MoveJ RelTool (starting_position, 122, -10.9, -364 \Rx:=2.5, \Ry:=-2.1, \Rz:=0), v200, z200, Tooldata_7;
MoveJ RelTool (starting_position, 122, -11.6, -364 \Rx:=2.5, \Ry:=-2.1, \Rz:=0), v200, z200, Tooldata_7;
MoveJ RelTool (starting_position, 121, -12.4, -364 \Rx:=2.6, \Ry:=-2.1, \Rz:=0), v200, z200, Tooldata_7;
MoveJ RelTool (starting_position, 120, -13.1, -364 \Rx:=2.6, \Ry:=-2.4, \Rz:=0), v200, z200, Tooldata_7;
MoveJ RelTool (starting_position, 119, -13.8, -364 \Rx:=2.7, \Ry:=-2.4, \Rz:=0), v200, z200, Tooldata_7;
MoveJ RelTool (starting_position, 119, -14.6, -363 \Rx:=2.8, \Ry:=-2.7, \Rz:=0), v200, z200, Tooldata_7;
MoveJ RelTool (starting_position, 118, -15.4, -363 \Rx:=3, \Ry:=-2.7, \Rz:=0), v200, z200, Tooldata_7;
MoveJ RelTool (starting_position, 117, -16.1, -363 \Rx:=3.2, \Ry:=-3, \Rz:=0), v200, z200, Tooldata_7;
MoveJ RelTool (starting_position, 116, -16.9, -363 \Rx:=3.4, \Ry:=-3, \Rz:=0), v200, z200, Tooldata_7;
MoveJ RelTool (starting_position, 115, -17.6, -363 \Rx:=3.6, \Ry:=-3.3, \Rz:=0), v200, z200, Tooldata_7;
MoveJ RelTool (starting_position, 114, -18.3, -363 \Rx:=3.8, \Ry:=-3.3, \Rz:=0), v200, z200, Tooldata_7;
MoveJ RelTool (starting_position, 113, -19.1, -363 \Rx:=4.1, \Ry:=-3.6, \Rz:=0), v200, z200, Tooldata_7;
MoveJ RelTool (starting_position, 112, -19.8, -363 \Rx:=4.3, \Ry:=-3.9, \Rz:=0), v200, z200, Tooldata_7;
MoveJ RelTool (starting_position, 111, -20.5, -362 \Rx:=4.6, \Ry:=-3.9, \Rz:=0), v200, z200, Tooldata_7;
MoveJ RelTool (starting_position, 110, -21.1, -362 \Rx:=4.8, \Ry:=-4.2, \Rz:=0), v200, z200, Tooldata_7;
MoveJ RelTool (starting_position, 109, -21.8, -362 \Rx:=5, \Ry:=-4.2, \Rz:=0), v200, z200, Tooldata_7;
MoveJ RelTool (starting_position, 108, -22.4, -362 \Rx:=5.2, \Ry:=-4.5, \Rz:=0), v200, z200, Tooldata_7;
MoveJ RelTool (starting_position, 107, -23, -361 \Rx:=5.5, \Ry:=-4.5, \Rz:=0), v200, z200, Tooldata_7;
MoveJ RelTool (starting_position, 107, -23.6, -361 \Rx:=5.6, \Ry:=-4.8, \Rz:=0), v200, z200, Tooldata_7;
MoveJ RelTool (starting_position, 106, -24.1, -360 \Rx:=5.8, \Ry:=-4.8, \Rz:=0), v200, z200, Tooldata_7;
MoveJ RelTool (starting_position, 105, -24.6, -360 \Rx:=5.9, \Ry:=-5.1, \Rz:=0), v200, z200, Tooldata_7;
MoveJ RelTool (starting_position, 104, -25.1, -359 \Rx:=6, \Ry:=-5.1, \Rz:=0), v200, z200, Tooldata_7;
MoveJ RelTool (starting_position, 103, -25.6, -359 \Rx:=6.2, \Ry:=-5.4, \Rz:=0), v200, z200, Tooldata_7;
MoveJ RelTool (starting_position, 103, -26, -358 \Rx:=6.3, \Ry:=-5.4, \Rz:=0), v200, z200, Tooldata_7;
MoveJ RelTool (starting_position, 103, -26.4, -357 \Rx:=6.4, \Ry:=-5.4, \Rz:=0), v200, z200, Tooldata_7;
MoveJ RelTool (starting_position, 103, -26.8, -356 \Rx:=6.5, \Ry:=-5.4, \Rz:=0), v200, z200, Tooldata_7;
MoveJ RelTool (starting_position, 103, -27.1, -355 \Rx:=6.6, \Ry:=-5.4, \Rz:=0), v200, z200, Tooldata_7;
MoveJ RelTool (starting_position, 103, -27.5, -354 \Rx:=6.7, \Ry:=-5.4, \Rz:=0), v200, z200, Tooldata_7;
MoveJ RelTool (starting_position, 103, -27.8, -353 \Rx:=6.8, \Ry:=-5.4, \Rz:=0), v200, z200, Tooldata_7;
MoveJ RelTool (starting_position, 103, -28.2, -352 \Rx:=6.9, \Ry:=-5.4, \Rz:=0), v200, z200, Tooldata_7;
MoveJ RelTool (starting_position, 104, -28.5, -351 \Rx:=7, \Ry:=-5.1, \Rz:=0), v200, z200, Tooldata_7;
MoveJ RelTool (starting_position, 105, -28.8, -350 \Rx:=7.1, \Ry:=-5.1, \Rz:=0), v200, z200, Tooldata_7;
MoveJ RelTool (starting_position, 106, -29, -349 \Rx:=7.2, \Ry:=-4.8, \Rz:=0), v200, z200, Tooldata_7;
MoveJ RelTool (starting_position, 108, -29.3, -348 \Rx:=7.4, \Ry:=-4.5, \Rz:=0), v200, z200, Tooldata_7;
MoveJ RelTool (starting_position, 109, -29.6, -347 \Rx:=7.6, \Ry:=-4.2, \Rz:=0), v200, z200, Tooldata_7;
MoveJ RelTool (starting_position, 111, -29.8, -346 \Rx:=7.8, \Ry:=-3.9, \Rz:=0), v200, z200, Tooldata_7;
MoveJ RelTool (starting_position, 113, -30.1, -345 \Rx:=8.1, \Ry:=-3.6, \Rz:=0), v200, z200, Tooldata_7;
MoveJ RelTool (starting_position, 115, -30.4, -344 \Rx:=8.4, \Ry:=-3.3, \Rz:=0), v200, z200, Tooldata_7;
MoveJ RelTool (starting_position, 117, -30.6, -343 \Rx:=8.7, \Ry:=-3, \Rz:=0), v200, z200, Tooldata_7;
MoveJ RelTool (starting_position, 119, -30.9, -343 \Rx:=8.9, \Ry:=-2.7, \Rz:=0), v200, z200, Tooldata_7;
MoveJ RelTool (starting_position, 121, -31.2, -342 \Rx:=9.2, \Ry:=-2.1, \Rz:=0), v200, z200, Tooldata_7;
MoveJ RelTool (starting_position, 123, -31.5, -342 \Rx:=9.5, \Ry:=-1.8, \Rz:=0), v200, z200, Tooldata_7;
MoveJ RelTool (starting_position, 126, -31.8, -341 \Rx:=9.7, \Ry:=-1.5, \Rz:=0), v200, z200, Tooldata_7;
MoveJ RelTool (starting_position, 128, -32.1, -341 \Rx:=10, \Ry:=-0.9, \Rz:=0), v200, z200, Tooldata_7;
MoveJ RelTool (starting_position, 131, -32.4, -341 \Rx:=10.3, \Ry:=-0.6, \Rz:=0), v200, z200, Tooldata_7;
MoveJ RelTool (starting_position, 134, -32.8, -341 \Rx:=10.6, \Ry:=-0, \Rz:=0), v200, z200, Tooldata_7;
MoveJ RelTool (starting_position, 137, -33.2, -341 \Rx:=10.9, \Ry:=0.6, \Rz:=0), v200, z200, Tooldata_7;
MoveJ RelTool (starting_position, 139, -33.6, -341 \Rx:=11.1, \Ry:=0.9, \Rz:=0), v200, z200, Tooldata_7;
MoveJ RelTool (starting_position, 142, -34, -341 \Rx:=11.3, \Ry:=1.5, \Rz:=0), v200, z200, Tooldata_7;
MoveJ RelTool (starting_position, 145, -34.4, -341 \Rx:=11.5, \Ry:=2.1, \Rz:=0), v200, z200, Tooldata_7;
MoveJ RelTool (starting_position, 148, -34.8, -342 \Rx:=11.6, \Ry:=2.4, \Rz:=0), v200, z200, Tooldata_7;
MoveJ RelTool (starting_position, 150, -35.3, -342 \Rx:=11.8, \Ry:=3, \Rz:=0), v200, z200, Tooldata_7;
MoveJ RelTool (starting_position, 153, -35.9, -343 \Rx:=11.9, \Ry:=3.3, \Rz:=0), v200, z200, Tooldata_7;
MoveJ RelTool (starting_position, 155, -36.4, -344 \Rx:=12, \Ry:=3.6, \Rz:=0), v200, z200, Tooldata_7;
MoveJ RelTool (starting_position, 157, -37, -344 \Rx:=12, \Ry:=4.2, \Rz:=0), v200, z200, Tooldata_7;
MoveJ RelTool (starting_position, 159, -37.6, -345 \Rx:=12, \Ry:=4.5, \Rz:=0), v200, z200, Tooldata_7;
MoveJ RelTool (starting_position, 161, -38.2, -346 \Rx:=12, \Ry:=4.8, \Rz:=0), v200, z200, Tooldata_7;
MoveJ RelTool (starting_position, 163, -38.8, -347 \Rx:=12, \Ry:=5.1, \Rz:=0), v200, z200, Tooldata_7;
MoveJ RelTool (starting_position, 165, -39.5, -348 \Rx:=11.9, \Ry:=5.4, \Rz:=0), v200, z200, Tooldata_7;
MoveJ RelTool (starting_position, 167, -40.2, -349 \Rx:=11.8, \Ry:=5.7, \Rz:=0), v200, z200, Tooldata_7;
MoveJ RelTool (starting_position, 168, -40.9, -349 \Rx:=11.6, \Ry:=6, \Rz:=0), v200, z200, Tooldata_7;
MoveJ RelTool (starting_position, 170, -41.6, -350 \Rx:=11.4, \Ry:=6.3, \Rz:=0), v200, z200, Tooldata_7;
MoveJ RelTool (starting_position, 171, -42.4, -351 \Rx:=11.1, \Ry:=6.6, \Rz:=0), v200, z200, Tooldata_7;
MoveJ RelTool (starting_position, 172, -43.1, -352 \Rx:=10.8, \Ry:=6.6, \Rz:=0), v200, z200, Tooldata_7;
MoveJ RelTool (starting_position, 173, -43.8, -353 \Rx:=10.4, \Ry:=6.9, \Rz:=0), v200, z200, Tooldata_7;
MoveJ RelTool (starting_position, 173, -44.6, -354 \Rx:=10.1, \Ry:=6.9, \Rz:=0), v200, z200, Tooldata_7;
MoveJ RelTool (starting_position, 174, -45.4, -355 \Rx:=9.6, \Ry:=6.9, \Rz:=0), v200, z200, Tooldata_7;
MoveJ RelTool (starting_position, 174, -46.1, -356 \Rx:=9.1, \Ry:=6.9, \Rz:=0), v200, z200, Tooldata_7;
MoveJ RelTool (starting_position, 175, -46.9, -357 \Rx:=8.6, \Ry:=7.2, \Rz:=0), v200, z200, Tooldata_7;
MoveJ RelTool (starting_position, 175, -47.6, -357 \Rx:=8.1, \Ry:=7.2, \Rz:=0), v200, z200, Tooldata_7;
MoveJ RelTool (starting_position, 175, -48.3, -358 \Rx:=7.6, \Ry:=7.2, \Rz:=0), v200, z200, Tooldata_7;
MoveJ RelTool (starting_position, 175, -49.1, -359 \Rx:=7, \Ry:=7.2, \Rz:=0), v200, z200, Tooldata_7;
MoveJ RelTool (starting_position, 174, -49.8, -360 \Rx:=6.4, \Ry:=6.9, \Rz:=0), v200, z200, Tooldata_7;
MoveJ RelTool (starting_position, 174, -50.5, -361 \Rx:=5.8, \Ry:=6.9, \Rz:=0), v200, z200, Tooldata_7;
MoveJ RelTool (starting_position, 173, -51.1, -361 \Rx:=5.3, \Ry:=6.9, \Rz:=0), v200, z200, Tooldata_7;
MoveJ RelTool (starting_position, 172, -51.8, -362 \Rx:=4.7, \Ry:=6.6, \Rz:=0), v200, z200, Tooldata_7;
MoveJ RelTool (starting_position, 172, -52.4, -363 \Rx:=4.1, \Ry:=6.6, \Rz:=0), v200, z200, Tooldata_7;
MoveJ RelTool (starting_position, 171, -53, -364 \Rx:=3.6, \Ry:=6.6, \Rz:=0), v200, z200, Tooldata_7;
MoveJ RelTool (starting_position, 170, -53.6, -364 \Rx:=3.1, \Ry:=6.3, \Rz:=0), v200, z200, Tooldata_7;
MoveJ RelTool (starting_position, 169, -54.1, -365 \Rx:=2.6, \Ry:=6.3, \Rz:=0), v200, z200, Tooldata_7;
MoveJ RelTool (starting_position, 168, -54.6, -366 \Rx:=2.2, \Ry:=6, \Rz:=0), v200, z200, Tooldata_7;
MoveJ RelTool (starting_position, 167, -55.1, -367 \Rx:=1.8, \Ry:=5.7, \Rz:=0), v200, z200, Tooldata_7;
MoveJ RelTool (starting_position, 165, -55.6, -367 \Rx:=1.4, \Ry:=5.4, \Rz:=0), v200, z200, Tooldata_7;
MoveJ RelTool (starting_position, 163, -56, -368 \Rx:=1, \Ry:=5.1, \Rz:=0), v200, z200, Tooldata_7;
MoveJ RelTool (starting_position, 162, -56.4, -369 \Rx:=0.7, \Ry:=4.8, \Rz:=0), v200, z200, Tooldata_7;
MoveJ RelTool (starting_position, 160, -56.8, -369 \Rx:=0.4, \Ry:=4.5, \Rz:=0), v200, z200, Tooldata_7;
MoveJ RelTool (starting_position, 158, -57.1, -370 \Rx:=0.2, \Ry:=4.2, \Rz:=0), v200, z200, Tooldata_7;
MoveJ RelTool (starting_position, 156, -57.5, -371 \Rx:=-0, \Ry:=3.9, \Rz:=0), v200, z200, Tooldata_7;
MoveJ RelTool (starting_position, 154, -57.8, -371 \Rx:=-0.2, \Ry:=3.6, \Rz:=0), v200, z200, Tooldata_7;
MoveJ RelTool (starting_position, 152, -58.1, -372 \Rx:=-0.3, \Ry:=3.3, \Rz:=0), v200, z200, Tooldata_7;
MoveJ RelTool (starting_position, 150, -58.4, -372 \Rx:=-0.4, \Ry:=2.7, \Rz:=0), v200, z200, Tooldata_7;
MoveJ RelTool (starting_position, 148, -58.7, -373 \Rx:=-0.4, \Ry:=2.4, \Rz:=0), v200, z200, Tooldata_7;
MoveJ RelTool (starting_position, 145, -59, -373 \Rx:=-0.4, \Ry:=2.1, \Rz:=0), v200, z200, Tooldata_7;
MoveJ RelTool (starting_position, 143, -59.2, -374 \Rx:=-0.4, \Ry:=1.5, \Rz:=0), v200, z200, Tooldata_7;
MoveJ RelTool (starting_position, 140, -59.5, -374 \Rx:=-0.4, \Ry:=1.2, \Rz:=0), v200, z200, Tooldata_7;
MoveJ RelTool (starting_position, 138, -59.7, -374 \Rx:=-0.4, \Ry:=0.6, \Rz:=0), v200, z200, Tooldata_7;
MoveJ RelTool (starting_position, 136, -60, -375 \Rx:=-0.4, \Ry:=0.3, \Rz:=0), v200, z200, Tooldata_7;
MoveJ RelTool (starting_position, 133, -60.2, -375 \Rx:=-0.3, \Ry:=-0, \Rz:=0), v200, z200, Tooldata_7;
MoveJ RelTool (starting_position, 131, -60.5, -375 \Rx:=-0.2, \Ry:=-0.6, \Rz:=0), v200, z200, Tooldata_7;
MoveJ RelTool (starting_position, 128, -60.7, -375 \Rx:=-0.1, \Ry:=-0.9, \Rz:=0), v200, z200, Tooldata_7;
MoveJ RelTool (starting_position, 126, -61, -375 \Rx:=0, \Ry:=-1.2, \Rz:=0), v200, z200, Tooldata_7;
MoveJ RelTool (starting_position, 123, -61.2, -374 \Rx:=0.1, \Ry:=-1.8, \Rz:=0), v200, z200, Tooldata_7;
MoveJ RelTool (starting_position, 121, -61.5, -374 \Rx:=0.2, \Ry:=-2.4, \Rz:=0), v200, z200, Tooldata_7;
MoveJ RelTool (starting_position, 118, -61.8, -374 \Rx:=0.3, \Ry:=-2.7, \Rz:=0), v200, z200, Tooldata_7;
MoveJ RelTool (starting_position, 116, -62.1, -373 \Rx:=0.4, \Ry:=-3, \Rz:=0), v200, z200, Tooldata_7;
MoveJ RelTool (starting_position, 113, -62.5, -373 \Rx:=0.4, \Ry:=-3.6, \Rz:=0), v200, z200, Tooldata_7;
MoveJ RelTool (starting_position, 111, -62.8, -372 \Rx:=0.5, \Ry:=-4.2, \Rz:=0), v200, z200, Tooldata_7;
MoveJ RelTool (starting_position, 109, -63.2, -372 \Rx:=0.6, \Ry:=-4.5, \Rz:=0), v200, z200, Tooldata_7;
MoveJ RelTool (starting_position, 107, -63.6, -371 \Rx:=0.6, \Ry:=-4.5, \Rz:=0), v200, z200, Tooldata_7;
MoveJ RelTool (starting_position, 105, -64, -371 \Rx:=0.6, \Ry:=-5.1, \Rz:=0), v200, z200, Tooldata_7;
MoveJ RelTool (starting_position, 103, -64.4, -370 \Rx:=0.6, \Ry:=-5.4, \Rz:=0), v200, z200, Tooldata_7;
MoveJ RelTool (starting_position, 101, -64.8, -369 \Rx:=0.5, \Ry:=-5.7, \Rz:=0), v200, z200, Tooldata_7;
MoveJ RelTool (starting_position, 99, -65.3, -368 \Rx:=0.4, \Ry:=-6, \Rz:=0), v200, z200, Tooldata_7;
MoveJ RelTool (starting_position, 98, -65.9, -368 \Rx:=0.3, \Ry:=-6.3, \Rz:=0), v200, z200, Tooldata_7;
MoveJ RelTool (starting_position, 96, -66.4, -367 \Rx:=0.2, \Ry:=-6.6, \Rz:=0), v200, z200, Tooldata_7;
MoveJ RelTool (starting_position, 95, -67, -366 \Rx:=0.1, \Ry:=-6.6, \Rz:=0), v200, z200, Tooldata_7;
MoveJ RelTool (starting_position, 94, -67.6, -365 \Rx:=-0.1, \Ry:=-6.9, \Rz:=0), v200, z200, Tooldata_7;
MoveJ RelTool (starting_position, 93, -68.2, -364 \Rx:=-0.4, \Ry:=-7.2, \Rz:=0), v200, z200, Tooldata_7;
MoveJ RelTool (starting_position, 92, -68.8, -363 \Rx:=-0.6, \Ry:=-7.2, \Rz:=0), v200, z200, Tooldata_7;
MoveJ RelTool (starting_position, 91, -69.5, -362 \Rx:=-0.9, \Ry:=-7.5, \Rz:=0), v200, z200, Tooldata_7;
MoveJ RelTool (starting_position, 90, -70.2, -362 \Rx:=-1.3, \Ry:=-7.5, \Rz:=0), v200, z200, Tooldata_7;
MoveJ RelTool (starting_position, 89, -70.9, -361 \Rx:=-1.6, \Ry:=-7.8, \Rz:=0), v200, z200, Tooldata_7;
MoveJ RelTool (starting_position, 89, -71.6, -360 \Rx:=-1.9, \Ry:=-7.8, \Rz:=0), v200, z200, Tooldata_7;
MoveJ RelTool (starting_position, 88, -72.4, -359 \Rx:=-2.3, \Ry:=-7.8, \Rz:=0), v200, z200, Tooldata_7;
MoveJ RelTool (starting_position, 88, -73.1, -358 \Rx:=-2.7, \Ry:=-8.1, \Rz:=0), v200, z200, Tooldata_7;
MoveJ RelTool (starting_position, 87, -73.8, -357 \Rx:=-3.1, \Ry:=-8.1, \Rz:=0), v200, z200, Tooldata_7;
MoveJ RelTool (starting_position, 87, -74.6, -356 \Rx:=-3.6, \Ry:=-8.1, \Rz:=0), v200, z200, Tooldata_7;
MoveJ RelTool (starting_position, 87, -75.4, -355 \Rx:=-4, \Ry:=-8.1, \Rz:=0), v200, z200, Tooldata_7;
MoveJ RelTool (starting_position, 87, -76.1, -354 \Rx:=-4.4, \Ry:=-8.4, \Rz:=0), v200, z200, Tooldata_7;
MoveJ RelTool (starting_position, 87, -76.9, -353 \Rx:=-4.8, \Ry:=-8.1, \Rz:=0), v200, z200, Tooldata_7;
MoveJ RelTool (starting_position, 87, -77.6, -352 \Rx:=-5.2, \Ry:=-8.1, \Rz:=0), v200, z200, Tooldata_7;
MoveJ RelTool (starting_position, 87, -78.3, -351 \Rx:=-5.6, \Ry:=-8.1, \Rz:=0), v200, z200, Tooldata_7;
MoveJ RelTool (starting_position, 88, -79.1, -351 \Rx:=-5.9, \Ry:=-8.1, \Rz:=0), v200, z200, Tooldata_7;
MoveJ RelTool (starting_position, 88, -79.8, -350 \Rx:=-6.2, \Ry:=-7.8, \Rz:=0), v200, z200, Tooldata_7;
MoveJ RelTool (starting_position, 88, -80.5, -349 \Rx:=-6.4, \Ry:=-7.8, \Rz:=0), v200, z200, Tooldata_7;
MoveJ RelTool (starting_position, 89, -81.1, -348 \Rx:=-6.6, \Ry:=-7.8, \Rz:=0), v200, z200, Tooldata_7;
MoveJ RelTool (starting_position, 90, -81.8, -347 \Rx:=-6.7, \Ry:=-7.8, \Rz:=0), v200, z200, Tooldata_7;
MoveJ RelTool (starting_position, 90, -82.4, -346 \Rx:=-6.8, \Ry:=-7.5, \Rz:=0), v200, z200, Tooldata_7;
MoveJ RelTool (starting_position, 91, -83, -345 \Rx:=-6.8, \Ry:=-7.5, \Rz:=0), v200, z200, Tooldata_7;
MoveJ RelTool (starting_position, 92, -83.6, -344 \Rx:=-6.7, \Ry:=-7.2, \Rz:=0), v200, z200, Tooldata_7;
MoveJ RelTool (starting_position, 93, -84.1, -343 \Rx:=-6.5, \Ry:=-7.2, \Rz:=0), v200, z200, Tooldata_7;
MoveJ RelTool (starting_position, 93, -84.6, -343 \Rx:=-6.3, \Ry:=-6.9, \Rz:=0), v200, z200, Tooldata_7;
MoveJ RelTool (starting_position, 94, -85.1, -342 \Rx:=-6.1, \Ry:=-6.9, \Rz:=0), v200, z200, Tooldata_7;
MoveJ RelTool (starting_position, 95, -85.6, -341 \Rx:=-5.7, \Ry:=-6.6, \Rz:=0), v200, z200, Tooldata_7;
MoveJ RelTool (starting_position, 96, -86, -340 \Rx:=-5.4, \Ry:=-6.6, \Rz:=0), v200, z200, Tooldata_7;
MoveJ RelTool (starting_position, 97, -86.4, -340 \Rx:=-5, \Ry:=-6.6, \Rz:=0), v200, z200, Tooldata_7;
MoveJ RelTool (starting_position, 97, -86.8, -339 \Rx:=-4.6, \Ry:=-6.3, \Rz:=0), v200, z200, Tooldata_7;
MoveJ RelTool (starting_position, 98, -87.1, -339 \Rx:=-4.1, \Ry:=-6, \Rz:=0), v200, z200, Tooldata_7;
MoveJ RelTool (starting_position, 99, -87.5, -338 \Rx:=-3.7, \Ry:=-6, \Rz:=0), v200, z200, Tooldata_7;
MoveJ RelTool (starting_position, 100, -87.7, -337 \Rx:=-3.3, \Ry:=-5.7, \Rz:=0), v200, z200, Tooldata_7;
MoveJ RelTool (starting_position, 101, -88, -337 \Rx:=-2.8, \Ry:=-5.7, \Rz:=0), v200, z200, Tooldata_7;
MoveJ RelTool (starting_position, 102, -88.3, -336 \Rx:=-2.4, \Ry:=-5.4, \Rz:=0), v200, z200, Tooldata_7;
MoveJ RelTool (starting_position, 102, -88.6, -336 \Rx:=-2, \Ry:=-5.4, \Rz:=0), v200, z200, Tooldata_7;
MoveJ RelTool (starting_position, 103, -88.8, -336 \Rx:=-1.7, \Ry:=-5.4, \Rz:=0), v200, z200, Tooldata_7;
MoveJ RelTool (starting_position, 103, -89.1, -335 \Rx:=-1.3, \Ry:=-5.4, \Rz:=0), v200, z200, Tooldata_7;
MoveJ RelTool (starting_position, 104, -89.3, -335 \Rx:=-1, \Ry:=-5.1, \Rz:=0), v200, z200, Tooldata_7;
MoveJ RelTool (starting_position, 104, -89.5, -335 \Rx:=-0.7, \Ry:=-5.1, \Rz:=0), v200, z200, Tooldata_7;
MoveJ RelTool (starting_position, 104, -89.7, -334 \Rx:=-0.5, \Ry:=-5.1, \Rz:=0), v200, z200, Tooldata_7;
MoveJ RelTool (starting_position, 104, -90, -334 \Rx:=-0.3, \Ry:=-5.1, \Rz:=0), v200, z200, Tooldata_7;
MoveJ RelTool (starting_position, 104, -90.2, -333 \Rx:=0, \Ry:=-5.1, \Rz:=0), v200, z200, Tooldata_7;
MoveJ RelTool (starting_position, 104, -90.4, -333 \Rx:=0.2, \Ry:=-5.1, \Rz:=0), v200, z200, Tooldata_7;
MoveJ RelTool (starting_position, 104, -90.6, -333 \Rx:=0.4, \Ry:=-5.1, \Rz:=0), v200, z200, Tooldata_7;
MoveJ RelTool (starting_position, 104, -90.9, -332 \Rx:=0.5, \Ry:=-5.1, \Rz:=0), v200, z200, Tooldata_7;
MoveJ RelTool (starting_position, 103, -91.1, -332 \Rx:=0.7, \Ry:=-5.4, \Rz:=0), v200, z200, Tooldata_7;
MoveJ RelTool (starting_position, 103, -91.4, -331 \Rx:=0.8, \Ry:=-5.4, \Rz:=0), v200, z200, Tooldata_7;
MoveJ RelTool (starting_position, 102, -91.6, -331 \Rx:=0.9, \Ry:=-5.4, \Rz:=0), v200, z200, Tooldata_7;
MoveJ RelTool (starting_position, 101, -91.9, -330 \Rx:=0.9, \Ry:=-5.7, \Rz:=0), v200, z200, Tooldata_7;
MoveJ RelTool (starting_position, 101, -92.2, -330 \Rx:=1, \Ry:=-5.7, \Rz:=0), v200, z200, Tooldata_7;
MoveJ RelTool (starting_position, 100, -92.5, -329 \Rx:=1, \Ry:=-6, \Rz:=0), v200, z200, Tooldata_7;
MoveJ RelTool (starting_position, 99, -92.8, -329 \Rx:=0.9, \Ry:=-6, \Rz:=0), v200, z200, Tooldata_7;
MoveJ RelTool (starting_position, 98, -93.2, -328 \Rx:=0.9, \Ry:=-6, \Rz:=0), v200, z200, Tooldata_7;
MoveJ RelTool (starting_position, 97, -93.6, -328 \Rx:=0.8, \Ry:=-6.3, \Rz:=0), v200, z200, Tooldata_7;
MoveJ RelTool (starting_position, 95, -94, -327 \Rx:=0.7, \Ry:=-6.6, \Rz:=0), v200, z200, Tooldata_7;
MoveJ RelTool (starting_position, 94, -94.4, -327 \Rx:=0.6, \Ry:=-6.9, \Rz:=0), v200, z200, Tooldata_7;
MoveJ RelTool (starting_position, 92, -94.8, -326 \Rx:=0.5, \Ry:=-7.2, \Rz:=0), v200, z200, Tooldata_7;
MoveJ RelTool (starting_position, 90, -95.3, -326 \Rx:=0.4, \Ry:=-7.5, \Rz:=0), v200, z200, Tooldata_7;
MoveJ RelTool (starting_position, 89, -95.9, -325 \Rx:=0.2, \Ry:=-7.8, \Rz:=0), v200, z200, Tooldata_7;
MoveJ RelTool (starting_position, 87, -96.4, -325 \Rx:=0.1, \Ry:=-8.1, \Rz:=0), v200, z200, Tooldata_7;
MoveJ RelTool (starting_position, 85, -97, -324 \Rx:=-0.1, \Ry:=-8.4, \Rz:=0), v200, z200, Tooldata_7;
MoveJ RelTool (starting_position, 83, -97.6, -323 \Rx:=-0.3, \Ry:=-9, \Rz:=0), v200, z200, Tooldata_7;
MoveJ RelTool (starting_position, 80, -98.2, -323 \Rx:=-0.5, \Ry:=-9.3, \Rz:=0), v200, z200, Tooldata_7;
MoveJ RelTool (starting_position, 78, -98.8, -322 \Rx:=-0.8, \Ry:=-9.6, \Rz:=0), v200, z200, Tooldata_7;
MoveJ RelTool (starting_position, 76, -99.5, -321 \Rx:=-1, \Ry:=-9.9, \Rz:=0), v200, z200, Tooldata_7;
MoveJ RelTool (starting_position, 74, -100.2, -320 \Rx:=-1.3, \Ry:=-10.5, \Rz:=0), v200, z200, Tooldata_7;
MoveJ RelTool (starting_position, 71, -100.9, -320 \Rx:=-1.5, \Ry:=-10.8, \Rz:=0), v200, z200, Tooldata_7;
MoveJ RelTool (starting_position, 68, -101.6, -319 \Rx:=-1.8, \Ry:=-11.4, \Rz:=0), v200, z200, Tooldata_7;
MoveJ RelTool (starting_position, 66, -102.4, -318 \Rx:=-2, \Ry:=-11.7, \Rz:=0), v200, z200, Tooldata_7;
MoveJ RelTool (starting_position, 63, -103.1, -317 \Rx:=-2.3, \Ry:=-12.3, \Rz:=0), v200, z200, Tooldata_7;
MoveJ RelTool (starting_position, 60, -103.8, -316 \Rx:=-2.5, \Ry:=-12.9, \Rz:=0), v200, z200, Tooldata_7;
MoveJ RelTool (starting_position, 57, -104.6, -315 \Rx:=-2.7, \Ry:=-13.5, \Rz:=0), v200, z200, Tooldata_7;
MoveJ RelTool (starting_position, 54, -105.4, -313 \Rx:=-2.9, \Ry:=-13.8, \Rz:=0), v200, z200, Tooldata_7;
MoveJ RelTool (starting_position, 51, -106.1, -312 \Rx:=-3.1, \Ry:=-14.4, \Rz:=0), v200, z200, Tooldata_7;
MoveJ RelTool (starting_position, 49, -106.9, -311 \Rx:=-3.1, \Ry:=-14.7, \Rz:=0), v200, z200, Tooldata_7;
MoveJ RelTool (starting_position, 46, -107.6, -309 \Rx:=-3.2, \Ry:=-15.3, \Rz:=0), v200, z200, Tooldata_7;
MoveJ RelTool (starting_position, 43, -108.3, -307 \Rx:=-3.2, \Ry:=-15.6, \Rz:=0), v200, z200, Tooldata_7;
MoveJ RelTool (starting_position, 41, -109.1, -306 \Rx:=-3.2, \Ry:=-16.2, \Rz:=0), v200, z200, Tooldata_7;
MoveJ RelTool (starting_position, 38, -109.8, -304 \Rx:=-3, \Ry:=-16.5, \Rz:=0), v200, z200, Tooldata_7;
MoveJ RelTool (starting_position, 36, -110.5, -302 \Rx:=-2.9, \Ry:=-17.1, \Rz:=0), v200, z200, Tooldata_7;
MoveJ RelTool (starting_position, 34, -111.1, -300 \Rx:=-2.8, \Ry:=-17.4, \Rz:=0), v200, z200, Tooldata_7;
MoveJ RelTool (starting_position, 32, -111.8, -298 \Rx:=-2.6, \Ry:=-17.7, \Rz:=0), v200, z200, Tooldata_7;
MoveJ RelTool (starting_position, 30, -112.4, -296 \Rx:=-2.3, \Ry:=-18, \Rz:=0), v200, z200, Tooldata_7;
MoveJ RelTool (starting_position, 28, -113, -294 \Rx:=-2, \Ry:=-18.3, \Rz:=0), v200, z200, Tooldata_7;
MoveJ RelTool (starting_position, 27, -113.6, -292 \Rx:=-1.7, \Ry:=-18.6, \Rz:=0), v200, z200, Tooldata_7;
MoveJ RelTool (starting_position, 26, -114.1, -290 \Rx:=-1.3, \Ry:=-18.9, \Rz:=0), v200, z200, Tooldata_7;
MoveJ RelTool (starting_position, 25, -114.6, -287 \Rx:=-0.9, \Ry:=-18.9, \Rz:=0), v200, z200, Tooldata_7;
MoveJ RelTool (starting_position, 24, -115.1, -285 \Rx:=-0.4, \Ry:=-19.2, \Rz:=0), v200, z200, Tooldata_7;
MoveJ RelTool (starting_position, 23, -115.6, -283 \Rx:=-0, \Ry:=-19.2, \Rz:=0), v200, z200, Tooldata_7;
MoveJ RelTool (starting_position, 23, -116, -280 \Rx:=0.4, \Ry:=-19.2, \Rz:=0), v200, z200, Tooldata_7;
MoveJ RelTool (starting_position, 23, -116.4, -278 \Rx:=0.9, \Ry:=-19.2, \Rz:=0), v200, z200, Tooldata_7;
MoveJ RelTool (starting_position, 23, -116.8, -275 \Rx:=1.3, \Ry:=-19.2, \Rz:=0), v200, z200, Tooldata_7;
MoveJ RelTool (starting_position, 23, -117.1, -273 \Rx:=1.7, \Ry:=-19.2, \Rz:=0), v200, z200, Tooldata_7;
MoveJ RelTool (starting_position, 24, -117.5, -271 \Rx:=2.2, \Ry:=-19.2, \Rz:=0), v200, z200, Tooldata_7;
MoveJ RelTool (starting_position, 24, -117.7, -268 \Rx:=2.6, \Ry:=-18.9, \Rz:=0), v200, z200, Tooldata_7;
MoveJ RelTool (starting_position, 25, -118, -266 \Rx:=3, \Ry:=-18.9, \Rz:=0), v200, z200, Tooldata_7;
MoveJ RelTool (starting_position, 26, -118.3, -263 \Rx:=3.4, \Ry:=-18.9, \Rz:=0), v200, z200, Tooldata_7;
MoveJ RelTool (starting_position, 27, -118.5, -261 \Rx:=3.9, \Ry:=-18.6, \Rz:=0), v200, z200, Tooldata_7;
MoveJ RelTool (starting_position, 28, -118.7, -259 \Rx:=4.2, \Ry:=-18.3, \Rz:=0), v200, z200, Tooldata_7;
MoveJ RelTool (starting_position, 30, -118.9, -257 \Rx:=4.6, \Ry:=-18, \Rz:=0), v200, z200, Tooldata_7;
MoveJ RelTool (starting_position, 32, -119.1, -254 \Rx:=4.9, \Ry:=-17.7, \Rz:=0), v200, z200, Tooldata_7;
MoveJ RelTool (starting_position, 33, -119.3, -252 \Rx:=5.2, \Ry:=-17.4, \Rz:=0), v200, z200, Tooldata_7;
MoveJ RelTool (starting_position, 35, -119.5, -250 \Rx:=5.5, \Ry:=-17.1, \Rz:=0), v200, z200, Tooldata_7;
MoveJ RelTool (starting_position, 37, -119.7, -249 \Rx:=5.6, \Ry:=-16.8, \Rz:=0), v200, z200, Tooldata_7;
MoveJ RelTool (starting_position, 39, -119.9, -247 \Rx:=5.7, \Ry:=-16.5, \Rz:=0), v200, z200, Tooldata_7;
MoveJ RelTool (starting_position, 41, -120.1, -245 \Rx:=5.8, \Ry:=-15.9, \Rz:=0), v200, z200, Tooldata_7;
MoveJ RelTool (starting_position, 43, -120.2, -243 \Rx:=5.8, \Ry:=-15.6, \Rz:=0), v200, z200, Tooldata_7;
MoveJ RelTool (starting_position, 45, -120.4, -242 \Rx:=5.8, \Ry:=-15.3, \Rz:=0), v200, z200, Tooldata_7;
MoveJ RelTool (starting_position, 47, -120.6, -240 \Rx:=5.8, \Ry:=-15, \Rz:=0), v200, z200, Tooldata_7;
MoveJ RelTool (starting_position, 49, -120.8, -239 \Rx:=5.7, \Ry:=-14.7, \Rz:=0), v200, z200, Tooldata_7;
MoveJ RelTool (starting_position, 51, -121, -238 \Rx:=5.6, \Ry:=-14.4, \Rz:=0), v200, z200, Tooldata_7;
MoveJ RelTool (starting_position, 53, -121.2, -236 \Rx:=5.5, \Ry:=-14.1, \Rz:=0), v200, z200, Tooldata_7;
MoveJ RelTool (starting_position, 55, -121.5, -235 \Rx:=5.3, \Ry:=-13.5, \Rz:=0), v200, z200, Tooldata_7;
MoveJ RelTool (starting_position, 57, -121.7, -234 \Rx:=5.2, \Ry:=-13.2, \Rz:=0), v200, z200, Tooldata_7;
MoveJ RelTool (starting_position, 59, -121.9, -233 \Rx:=5, \Ry:=-12.9, \Rz:=0), v200, z200, Tooldata_7;
MoveJ RelTool (starting_position, 60, -122.2, -232 \Rx:=4.8, \Ry:=-12.6, \Rz:=0), v200, z200, Tooldata_7;
MoveJ RelTool (starting_position, 61, -122.5, -231 \Rx:=4.5, \Ry:=-12.6, \Rz:=0), v200, z200, Tooldata_7;
MoveJ RelTool (starting_position, 63, -122.8, -230 \Rx:=4.3, \Ry:=-12.3, \Rz:=0), v200, z200, Tooldata_7;
MoveJ RelTool (starting_position, 64, -123.2, -230 \Rx:=4.1, \Ry:=-12, \Rz:=0), v200, z200, Tooldata_7;
MoveJ RelTool (starting_position, 65, -123.6, -229 \Rx:=3.9, \Ry:=-12, \Rz:=0), v200, z200, Tooldata_7;
MoveJ RelTool (starting_position, 66, -124, -228 \Rx:=3.6, \Ry:=-11.7, \Rz:=0), v200, z200, Tooldata_7;
MoveJ RelTool (starting_position, 67, -124.4, -227 \Rx:=3.5, \Ry:=-11.4, \Rz:=0), v200, z200, Tooldata_7;
MoveJ RelTool (starting_position, 68, -124.8, -226 \Rx:=3.3, \Ry:=-11.4, \Rz:=0), v200, z200, Tooldata_7;
MoveJ RelTool (starting_position, 68, -125.3, -225 \Rx:=3.2, \Ry:=-11.4, \Rz:=0), v200, z200, Tooldata_7;
MoveJ RelTool (starting_position, 69, -125.9, -224 \Rx:=3, \Ry:=-11.1, \Rz:=0), v200, z200, Tooldata_7;
MoveJ RelTool (starting_position, 69, -126.4, -223 \Rx:=3, \Ry:=-11.1, \Rz:=0), v200, z200, Tooldata_7;
MoveJ RelTool (starting_position, 69, -127, -222 \Rx:=3, \Ry:=-11.1, \Rz:=0), v200, z200, Tooldata_7;
MoveJ RelTool (starting_position, 70, -127.6, -221 \Rx:=3.1, \Ry:=-11.1, \Rz:=0), v200, z200, Tooldata_7;
MoveJ RelTool (starting_position, 70, -128.2, -220 \Rx:=3.2, \Ry:=-11.1, \Rz:=0), v200, z200, Tooldata_7;
MoveJ RelTool (starting_position, 70, -128.8, -219 \Rx:=3.3, \Ry:=-11.1, \Rz:=0), v200, z200, Tooldata_7;
MoveJ RelTool (starting_position, 70, -129.5, -218 \Rx:=3.5, \Ry:=-11.1, \Rz:=0), v200, z200, Tooldata_7;
MoveJ RelTool (starting_position, 70, -130.2, -217 \Rx:=3.7, \Ry:=-11.1, \Rz:=0), v200, z200, Tooldata_7;
MoveJ RelTool (starting_position, 70, -130.9, -216 \Rx:=3.9, \Ry:=-11.1, \Rz:=0), v200, z200, Tooldata_7;
MoveJ RelTool (starting_position, 70, -131.6, -214 \Rx:=4.1, \Ry:=-11.1, \Rz:=0), v200, z200, Tooldata_7;
MoveJ RelTool (starting_position, 70, -132.4, -213 \Rx:=4.3, \Ry:=-11.1, \Rz:=0), v200, z200, Tooldata_7;
MoveJ RelTool (starting_position, 70, -133.1, -212 \Rx:=4.6, \Ry:=-11.1, \Rz:=0), v200, z200, Tooldata_7;
MoveJ RelTool (starting_position, 70, -133.8, -211 \Rx:=4.8, \Ry:=-11.1, \Rz:=0), v200, z200, Tooldata_7;
MoveJ RelTool (starting_position, 69, -134.6, -209 \Rx:=5, \Ry:=-11.1, \Rz:=0), v200, z200, Tooldata_7;
MoveJ RelTool (starting_position, 69, -135.4, -208 \Rx:=5.3, \Ry:=-11.1, \Rz:=0), v200, z200, Tooldata_7;
MoveJ RelTool (starting_position, 69, -136.1, -207 \Rx:=5.5, \Ry:=-11.4, \Rz:=0), v200, z200, Tooldata_7;
MoveJ RelTool (starting_position, 69, -136.9, -206 \Rx:=5.7, \Ry:=-11.1, \Rz:=0), v200, z200, Tooldata_7;
MoveJ RelTool (starting_position, 69, -137.6, -204 \Rx:=5.9, \Ry:=-11.1, \Rz:=0), v200, z200, Tooldata_7;
MoveJ RelTool (starting_position, 69, -138.3, -203 \Rx:=6.1, \Ry:=-11.1, \Rz:=0), v200, z200, Tooldata_7;
MoveJ RelTool (starting_position, 68, -139.1, -202 \Rx:=6.3, \Ry:=-11.4, \Rz:=0), v200, z200, Tooldata_7;
MoveJ RelTool (starting_position, 68, -139.8, -201 \Rx:=6.4, \Ry:=-11.4, \Rz:=0), v200, z200, Tooldata_7;
MoveJ RelTool (starting_position, 67, -140.5, -199 \Rx:=6.5, \Ry:=-11.4, \Rz:=0), v200, z200, Tooldata_7;
MoveJ RelTool (starting_position, 67, -141.1, -198 \Rx:=6.5, \Ry:=-11.7, \Rz:=0), v200, z200, Tooldata_7;
MoveJ RelTool (starting_position, 66, -141.8, -197 \Rx:=6.5, \Ry:=-11.7, \Rz:=0), v200, z200, Tooldata_7;
MoveJ RelTool (starting_position, 65, -142.4, -196 \Rx:=6.5, \Ry:=-12, \Rz:=0), v200, z200, Tooldata_7;
MoveJ RelTool (starting_position, 64, -143, -195 \Rx:=6.4, \Ry:=-12, \Rz:=0), v200, z200, Tooldata_7;
MoveJ RelTool (starting_position, 63, -143.6, -194 \Rx:=6.4, \Ry:=-12.3, \Rz:=0), v200, z200, Tooldata_7;
MoveJ RelTool (starting_position, 62, -144.1, -193 \Rx:=6.2, \Ry:=-12.3, \Rz:=0), v200, z200, Tooldata_7;
MoveJ RelTool (starting_position, 61, -144.6, -191 \Rx:=6.1, \Ry:=-12.6, \Rz:=0), v200, z200, Tooldata_7;
MoveJ RelTool (starting_position, 59, -145.1, -190 \Rx:=6, \Ry:=-12.9, \Rz:=0), v200, z200, Tooldata_7;
MoveJ RelTool (starting_position, 57, -145.6, -189 \Rx:=5.7, \Ry:=-13.2, \Rz:=0), v200, z200, Tooldata_7;
MoveJ RelTool (starting_position, 56, -146, -188 \Rx:=5.5, \Ry:=-13.5, \Rz:=0), v200, z200, Tooldata_7;
MoveJ RelTool (starting_position, 53, -146.4, -187 \Rx:=5.2, \Ry:=-13.8, \Rz:=0), v200, z200, Tooldata_7;
MoveJ RelTool (starting_position, 51, -146.8, -186 \Rx:=4.8, \Ry:=-14.4, \Rz:=0), v200, z200, Tooldata_7;
MoveJ RelTool (starting_position, 50, -147.1, -185 \Rx:=4.4, \Ry:=-14.7, \Rz:=0), v200, z200, Tooldata_7;
MoveJ RelTool (starting_position, 48, -147.5, -184 \Rx:=4, \Ry:=-15, \Rz:=0), v200, z200, Tooldata_7;
MoveJ RelTool (starting_position, 46, -147.7, -183 \Rx:=3.5, \Ry:=-15.3, \Rz:=0), v200, z200, Tooldata_7;
MoveJ RelTool (starting_position, 45, -148, -182 \Rx:=3, \Ry:=-15.3, \Rz:=0), v200, z200, Tooldata_7;
MoveJ RelTool (starting_position, 43, -148.3, -181 \Rx:=2.5, \Ry:=-15.6, \Rz:=0), v200, z200, Tooldata_7;
MoveJ RelTool (starting_position, 42, -148.5, -180 \Rx:=2.1, \Ry:=-15.9, \Rz:=0), v200, z200, Tooldata_7;
MoveJ RelTool (starting_position, 40, -148.7, -178 \Rx:=1.6, \Ry:=-16.2, \Rz:=0), v200, z200, Tooldata_7;
MoveJ RelTool (starting_position, 39, -148.9, -177 \Rx:=1.1, \Ry:=-16.5, \Rz:=0), v200, z200, Tooldata_7;
MoveJ RelTool (starting_position, 37, -149, -176 \Rx:=0.6, \Ry:=-16.8, \Rz:=0), v200, z200, Tooldata_7;
MoveJ RelTool (starting_position, 35, -149.2, -174 \Rx:=0.1, \Ry:=-17.1, \Rz:=0), v200, z200, Tooldata_7;
MoveJ RelTool (starting_position, 33, -149.4, -173 \Rx:=-0.4, \Ry:=-17.4, \Rz:=0), v200, z200, Tooldata_7;
MoveJ RelTool (starting_position, 30, -149.5, -171 \Rx:=-0.8, \Ry:=-18, \Rz:=0), v200, z200, Tooldata_7;
MoveJ RelTool (starting_position, 28, -149.7, -169 \Rx:=-1.3, \Ry:=-18.3, \Rz:=0), v200, z200, Tooldata_7;
MoveJ RelTool (starting_position, 25, -149.8, -167 \Rx:=-1.7, \Ry:=-18.9, \Rz:=0), v200, z200, Tooldata_7;
MoveJ RelTool (starting_position, 23, -150, -165 \Rx:=-2.1, \Ry:=-19.2, \Rz:=0), v200, z200, Tooldata_7;
MoveJ RelTool (starting_position, 21, -150.1, -163 \Rx:=-2.5, \Ry:=-19.8, \Rz:=0), v200, z200, Tooldata_7;
MoveJ RelTool (starting_position, 20, -150.3, -160 \Rx:=-3, \Ry:=-20.1, \Rz:=0), v200, z200, Tooldata_7;
MoveJ RelTool (starting_position, 19, -150.4, -158 \Rx:=-3.5, \Ry:=-20.1, \Rz:=0), v200, z200, Tooldata_7;
MoveJ RelTool (starting_position, 18, -150.6, -155 \Rx:=-3.9, \Ry:=-20.1, \Rz:=0), v200, z200, Tooldata_7;
MoveJ RelTool (starting_position, 18, -150.8, -152 \Rx:=-4.4, \Ry:=-20.1, \Rz:=0), v200, z200, Tooldata_7;
MoveJ RelTool (starting_position, 18, -150.9, -150 \Rx:=-4.8, \Ry:=-20.1, \Rz:=0), v200, z200, Tooldata_7;
MoveJ RelTool (starting_position, 19, -151.1, -147 \Rx:=-5.2, \Ry:=-20.1, \Rz:=0), v200, z200, Tooldata_7;
MoveJ RelTool (starting_position, 20, -151.3, -144 \Rx:=-5.4, \Ry:=-19.8, \Rz:=0), v200, z200, Tooldata_7;
MoveJ RelTool (starting_position, 22, -151.5, -142 \Rx:=-5.8, \Ry:=-19.5, \Rz:=0), v200, z200, Tooldata_7;
MoveJ RelTool (starting_position, 24, -151.7, -139 \Rx:=-6.1, \Ry:=-19.2, \Rz:=0), v200, z200, Tooldata_7;
MoveJ RelTool (starting_position, 26, -151.9, -137 \Rx:=-6.3, \Ry:=-18.9, \Rz:=0), v200, z200, Tooldata_7;
MoveJ RelTool (starting_position, 29, -152.2, -135 \Rx:=-6.5, \Ry:=-18.3, \Rz:=0), v200, z200, Tooldata_7;
MoveJ RelTool (starting_position, 32, -152.5, -132 \Rx:=-6.6, \Ry:=-17.7, \Rz:=0), v200, z200, Tooldata_7;
MoveJ RelTool (starting_position, 36, -152.8, -130 \Rx:=-6.7, \Ry:=-17.1, \Rz:=0), v200, z200, Tooldata_7;
MoveJ RelTool (starting_position, 40, -153.2, -128 \Rx:=-6.8, \Ry:=-16.5, \Rz:=0), v200, z200, Tooldata_7;
MoveJ RelTool (starting_position, 44, -153.6, -127 \Rx:=-6.9, \Ry:=-15.6, \Rz:=0), v200, z200, Tooldata_7;
MoveJ RelTool (starting_position, 49, -154, -125 \Rx:=-6.9, \Ry:=-14.7, \Rz:=0), v200, z200, Tooldata_7;
MoveJ RelTool (starting_position, 54, -154.4, -124 \Rx:=-6.8, \Ry:=-13.8, \Rz:=0), v200, z200, Tooldata_7;
MoveJ RelTool (starting_position, 59, -154.8, -123 \Rx:=-6.7, \Ry:=-12.9, \Rz:=0), v200, z200, Tooldata_7;
MoveJ RelTool (starting_position, 65, -155.3, -122 \Rx:=-6.6, \Ry:=-12, \Rz:=0), v200, z200, Tooldata_7;
MoveJ RelTool (starting_position, 71, -155.9, -121 \Rx:=-6.4, \Ry:=-10.8, \Rz:=0), v200, z200, Tooldata_7;
MoveJ RelTool (starting_position, 77, -156.4, -121 \Rx:=-6.2, \Ry:=-9.9, \Rz:=0), v200, z200, Tooldata_7;
MoveJ RelTool (starting_position, 84, -157, -121 \Rx:=-6, \Ry:=-8.7, \Rz:=0), v200, z200, Tooldata_7;
MoveJ RelTool (starting_position, 90, -157.6, -121 \Rx:=-5.8, \Ry:=-7.5, \Rz:=0), v200, z200, Tooldata_7;
MoveJ RelTool (starting_position, 97, -158.2, -121 \Rx:=-5.5, \Ry:=-6.3, \Rz:=0), v200, z200, Tooldata_7;
MoveJ RelTool (starting_position, 104, -158.8, -121 \Rx:=-5.2, \Ry:=-5.1, \Rz:=0), v200, z200, Tooldata_7;
MoveJ RelTool (starting_position, 111, -159.5, -122 \Rx:=-4.9, \Ry:=-3.9, \Rz:=0), v200, z200, Tooldata_7;
MoveJ RelTool (starting_position, 118, -160.2, -122 \Rx:=-4.5, \Ry:=-2.7, \Rz:=0), v200, z200, Tooldata_7;
MoveJ RelTool (starting_position, 125, -160.9, -121 \Rx:=-4.1, \Ry:=-1.5, \Rz:=0), v200, z200, Tooldata_7;
MoveJ RelTool (starting_position, 131, -161.6, -121 \Rx:=-3.7, \Ry:=-0.3, \Rz:=0), v200, z200, Tooldata_7;
MoveJ RelTool (starting_position, 138, -162.4, -120 \Rx:=-3.3, \Ry:=0.9, \Rz:=0), v200, z200, Tooldata_7;
MoveJ RelTool (starting_position, 144, -163.1, -119 \Rx:=-2.8, \Ry:=1.8, \Rz:=0), v200, z200, Tooldata_7;
MoveJ RelTool (starting_position, 151, -163.8, -118 \Rx:=-2.2, \Ry:=3, \Rz:=0), v200, z200, Tooldata_7;
MoveJ RelTool (starting_position, 157, -164.6, -116 \Rx:=-1.6, \Ry:=4.2, \Rz:=0), v200, z200, Tooldata_7;
MoveJ RelTool (starting_position, 163, -165.4, -114 \Rx:=-0.9, \Ry:=5.1, \Rz:=0), v200, z200, Tooldata_7;
MoveJ RelTool (starting_position, 168, -166.1, -112 \Rx:=-0.2, \Ry:=6, \Rz:=0), v200, z200, Tooldata_7;
MoveJ RelTool (starting_position, 174, -166.9, -109 \Rx:=0.6, \Ry:=7.2, \Rz:=0), v200, z200, Tooldata_7;
MoveJ RelTool (starting_position, 179, -167.6, -106 \Rx:=1.4, \Ry:=8.1, \Rz:=0), v200, z200, Tooldata_7;
MoveJ RelTool (starting_position, 184, -168.3, -103 \Rx:=2.2, \Ry:=8.7, \Rz:=0), v200, z200, Tooldata_7;
MoveJ RelTool (starting_position, 188, -169.1, -100 \Rx:=3, \Ry:=9.6, \Rz:=0), v200, z200, Tooldata_7;
MoveJ RelTool (starting_position, 192, -169.8, -97 \Rx:=3.9, \Ry:=10.2, \Rz:=0), v200, z200, Tooldata_7;
MoveJ RelTool (starting_position, 196, -170.5, -94 \Rx:=4.7, \Ry:=10.8, \Rz:=0), v200, z200, Tooldata_7;
MoveJ RelTool (starting_position, 199, -171.1, -92 \Rx:=5.6, \Ry:=11.4, \Rz:=0), v200, z200, Tooldata_7;
MoveJ RelTool (starting_position, 202, -171.8, -89 \Rx:=6.5, \Ry:=12, \Rz:=0), v200, z200, Tooldata_7;
MoveJ RelTool (starting_position, 204, -172.4, -87 \Rx:=7.3, \Ry:=12.3, \Rz:=0), v200, z200, Tooldata_7;
MoveJ RelTool (starting_position, 206, -173, -85 \Rx:=8.1, \Ry:=12.6, \Rz:=0), v200, z200, Tooldata_7;
MoveJ RelTool (starting_position, 208, -173.6, -83 \Rx:=8.8, \Ry:=13.2, \Rz:=0), v200, z200, Tooldata_7;
MoveJ RelTool (starting_position, 209, -174.1, -82 \Rx:=9.4, \Ry:=13.2, \Rz:=0), v200, z200, Tooldata_7;
MoveJ RelTool (starting_position, 210, -174.6, -81 \Rx:=10, \Ry:=13.2, \Rz:=0), v200, z200, Tooldata_7;
MoveJ RelTool (starting_position, 211, -175.1, -81 \Rx:=10.5, \Ry:=13.5, \Rz:=0), v200, z200, Tooldata_7;
MoveJ RelTool (starting_position, 211, -175.6, -80 \Rx:=11, \Ry:=13.5, \Rz:=0), v200, z200, Tooldata_7;
MoveJ RelTool (starting_position, 211, -176, -80 \Rx:=11.4, \Ry:=13.5, \Rz:=0), v200, z200, Tooldata_7;
MoveJ RelTool (starting_position, 211, -176.4, -81 \Rx:=11.7, \Ry:=13.5, \Rz:=0), v200, z200, Tooldata_7;
MoveJ RelTool (starting_position, 211, -176.8, -81 \Rx:=11.9, \Ry:=13.5, \Rz:=0), v200, z200, Tooldata_7;
MoveJ RelTool (starting_position, 210, -177.1, -81 \Rx:=12.1, \Ry:=13.2, \Rz:=0), v200, z200, Tooldata_7;
MoveJ RelTool (starting_position, 209, -177.5, -82 \Rx:=12.2, \Ry:=13.2, \Rz:=0), v200, z200, Tooldata_7;
MoveJ RelTool (starting_position, 208, -177.7, -83 \Rx:=12.2, \Ry:=12.9, \Rz:=0), v200, z200, Tooldata_7;
MoveJ RelTool (starting_position, 206, -178, -84 \Rx:=12.1, \Ry:=12.6, \Rz:=0), v200, z200, Tooldata_7;
MoveJ RelTool (starting_position, 204, -178.3, -85 \Rx:=12.1, \Ry:=12.3, \Rz:=0), v200, z200, Tooldata_7;
MoveJ RelTool (starting_position, 202, -178.5, -86 \Rx:=12, \Ry:=11.7, \Rz:=0), v200, z200, Tooldata_7;
MoveJ RelTool (starting_position, 199, -178.7, -87 \Rx:=11.8, \Ry:=11.4, \Rz:=0), v200, z200, Tooldata_7;
MoveJ RelTool (starting_position, 196, -178.9, -88 \Rx:=11.6, \Ry:=10.8, \Rz:=0), v200, z200, Tooldata_7;
MoveJ RelTool (starting_position, 194, -179, -89 \Rx:=11.5, \Ry:=10.5, \Rz:=0), v200, z200, Tooldata_7;
MoveJ RelTool (starting_position, 191, -179.2, -90 \Rx:=11.3, \Ry:=9.9, \Rz:=0), v200, z200, Tooldata_7;
MoveJ RelTool (starting_position, 187, -179.3, -91 \Rx:=11.1, \Ry:=9.3, \Rz:=0), v200, z200, Tooldata_7;
MoveJ RelTool (starting_position, 184, -179.4, -92 \Rx:=10.8, \Ry:=8.7, \Rz:=0), v200, z200, Tooldata_7;
MoveJ RelTool (starting_position, 180, -179.5, -93 \Rx:=10.6, \Ry:=8.1, \Rz:=0), v200, z200, Tooldata_7;
MoveJ RelTool (starting_position, 175, -179.6, -94 \Rx:=10.4, \Ry:=7.2, \Rz:=0), v200, z200, Tooldata_7;
MoveJ RelTool (starting_position, 171, -179.7, -95 \Rx:=10.2, \Ry:=6.3, \Rz:=0), v200, z200, Tooldata_7;
MoveJ RelTool (starting_position, 167, -179.8, -96 \Rx:=10, \Ry:=5.7, \Rz:=0), v200, z200, Tooldata_7;
MoveJ RelTool (starting_position, 162, -179.9, -96 \Rx:=9.9, \Ry:=4.8, \Rz:=0), v200, z200, Tooldata_7;
MoveJ RelTool (starting_position, 158, -180, -97 \Rx:=9.8, \Ry:=4.2, \Rz:=0), v200, z200, Tooldata_7;
MoveJ RelTool (starting_position, 154, -180.1, -97 \Rx:=9.8, \Ry:=3.3, \Rz:=0), v200, z200, Tooldata_7;
MoveJ RelTool (starting_position, 150, -180.2, -97 \Rx:=9.7, \Ry:=2.7, \Rz:=0), v200, z200, Tooldata_7;
MoveJ RelTool (starting_position, 146, -180.3, -98 \Rx:=9.7, \Ry:=1.8, \Rz:=0), v200, z200, Tooldata_7;
MoveJ RelTool (starting_position, 142, -180.3, -98 \Rx:=9.6, \Ry:=1.5, \Rz:=0), v200, z200, Tooldata_7;
MoveJ RelTool (starting_position, 138, -180.4, -98 \Rx:=9.6, \Ry:=0.9, \Rz:=0), v200, z200, Tooldata_7;
MoveJ RelTool (starting_position, 134, -180.5, -98 \Rx:=9.5, \Ry:=0, \Rz:=0), v200, z200, Tooldata_7;
MoveJ RelTool (starting_position, 131, -180.7, -98 \Rx:=9.4, \Ry:=-0.6, \Rz:=0), v200, z200, Tooldata_7;
MoveJ RelTool (starting_position, 127, -180.8, -98 \Rx:=9.3, \Ry:=-1.2, \Rz:=0), v200, z200, Tooldata_7;
MoveJ RelTool (starting_position, 122, -180.9, -98 \Rx:=9.1, \Ry:=-1.8, \Rz:=0), v200, z200, Tooldata_7;
MoveJ RelTool (starting_position, 118, -181.1, -98 \Rx:=8.9, \Ry:=-2.7, \Rz:=0), v200, z200, Tooldata_7;
MoveJ RelTool (starting_position, 113, -181.3, -98 \Rx:=8.6, \Ry:=-3.6, \Rz:=0), v200, z200, Tooldata_7;
MoveJ RelTool (starting_position, 108, -181.5, -97 \Rx:=8.2, \Ry:=-4.5, \Rz:=0), v200, z200, Tooldata_7;
MoveJ RelTool (starting_position, 103, -181.7, -97 \Rx:=7.8, \Ry:=-5.4, \Rz:=0), v200, z200, Tooldata_7;
MoveJ RelTool (starting_position, 98, -181.9, -96 \Rx:=7.4, \Ry:=-6.3, \Rz:=0), v200, z200, Tooldata_7;
MoveJ RelTool (starting_position, 92, -182.2, -96 \Rx:=6.8, \Ry:=-7.2, \Rz:=0), v200, z200, Tooldata_7;
MoveJ RelTool (starting_position, 87, -182.5, -95 \Rx:=6.3, \Ry:=-8.1, \Rz:=0), v200, z200, Tooldata_7;
MoveJ RelTool (starting_position, 82, -182.8, -95 \Rx:=5.8, \Ry:=-9, \Rz:=0), v200, z200, Tooldata_7;
MoveJ RelTool (starting_position, 77, -183.2, -94 \Rx:=5.1, \Ry:=-9.9, \Rz:=0), v200, z200, Tooldata_7;
MoveJ RelTool (starting_position, 72, -183.6, -93 \Rx:=4.4, \Ry:=-10.8, \Rz:=0), v200, z200, Tooldata_7;
MoveJ RelTool (starting_position, 66, -184, -92 \Rx:=3.7, \Ry:=-11.7, \Rz:=0), v200, z200, Tooldata_7;
MoveJ RelTool (starting_position, 61, -184.4, -91 \Rx:=2.9, \Ry:=-12.6, \Rz:=0), v200, z200, Tooldata_7;
MoveJ RelTool (starting_position, 56, -184.8, -90 \Rx:=2.2, \Ry:=-13.5, \Rz:=0), v200, z200, Tooldata_7;
MoveJ RelTool (starting_position, 51, -185.3, -89 \Rx:=1.5, \Ry:=-14.4, \Rz:=0), v200, z200, Tooldata_7;
MoveJ RelTool (starting_position, 46, -185.9, -87 \Rx:=0.8, \Ry:=-15.3, \Rz:=0), v200, z200, Tooldata_7;
MoveJ RelTool (starting_position, 41, -186.4, -86 \Rx:=0.2, \Ry:=-16.2, \Rz:=0), v200, z200, Tooldata_7;
MoveJ RelTool (starting_position, 36, -187, -84 \Rx:=-0.3, \Ry:=-16.8, \Rz:=0), v200, z200, Tooldata_7;
MoveJ RelTool (starting_position, 30, -187.6, -82 \Rx:=-0.8, \Ry:=-18, \Rz:=0), v200, z200, Tooldata_7;
MoveJ RelTool (starting_position, 25, -188.2, -81 \Rx:=-1.3, \Ry:=-18.9, \Rz:=0), v200, z200, Tooldata_7;
MoveJ RelTool (starting_position, 19, -188.8, -79 \Rx:=-1.6, \Ry:=-19.8, \Rz:=0), v200, z200, Tooldata_7;
MoveJ RelTool (starting_position, 14, -189.5, -77 \Rx:=-1.9, \Ry:=-20.7, \Rz:=0), v200, z200, Tooldata_7;
MoveJ RelTool (starting_position, 8, -190.2, -75 \Rx:=-2.1, \Ry:=-21.9, \Rz:=0), v200, z200, Tooldata_7;
MoveJ RelTool (starting_position, 2, -190.9, -72 \Rx:=-2.3, \Ry:=-22.8, \Rz:=0), v200, z200, Tooldata_7;
MoveJ RelTool (starting_position, -4, -191.6, -70 \Rx:=-2.4, \Ry:=-24, \Rz:=0), v200, z200, Tooldata_7;
MoveJ RelTool (starting_position, -10, -192.4, -67 \Rx:=-2.3, \Ry:=-24.9, \Rz:=0), v200, z200, Tooldata_7;
MoveJ RelTool (starting_position, -16, -193.1, -64 \Rx:=-2.1, \Ry:=-26.1, \Rz:=0), v200, z200, Tooldata_7;
MoveJ RelTool (starting_position, -21, -193.8, -62 \Rx:=-1.9, \Ry:=-27, \Rz:=0), v200, z200, Tooldata_7;
MoveJ RelTool (starting_position, -26, -194.6, -59 \Rx:=-1.6, \Ry:=-27.9, \Rz:=0), v200, z200, Tooldata_7;
MoveJ RelTool (starting_position, -30, -195.4, -56 \Rx:=-1.2, \Ry:=-28.5, \Rz:=0), v200, z200, Tooldata_7;
MoveJ RelTool (starting_position, -34, -196.1, -52 \Rx:=-0.8, \Ry:=-29.1, \Rz:=0), v200, z200, Tooldata_7;
MoveJ RelTool (starting_position, -38, -196.9, -49 \Rx:=-0.4, \Ry:=-29.7, \Rz:=0), v200, z200, Tooldata_7;
MoveJ RelTool (starting_position, -41, -197.6, -46 \Rx:=0.1, \Ry:=-30.6, \Rz:=0), v200, z200, Tooldata_7;
MoveJ RelTool (starting_position, -45, -198.3, -42 \Rx:=0.6, \Ry:=-30.9, \Rz:=0), v200, z200, Tooldata_7;
MoveJ RelTool (starting_position, -48, -199.1, -39 \Rx:=1.1, \Ry:=-31.5, \Rz:=0), v200, z200, Tooldata_7;
MoveJ RelTool (starting_position, -50, -199.8, -35 \Rx:=1.7, \Ry:=-32.1, \Rz:=0), v200, z200, Tooldata_7;
MoveJ RelTool (starting_position, -52, -200.5, -31 \Rx:=2.3, \Ry:=-32.4, \Rz:=0), v200, z200, Tooldata_7;
MoveJ RelTool (starting_position, -53, -201.1, -27 \Rx:=2.8, \Ry:=-32.7, \Rz:=0), v200, z200, Tooldata_7;
MoveJ RelTool (starting_position, -54, -201.8, -23 \Rx:=3.4, \Ry:=-32.7, \Rz:=0), v200, z200, Tooldata_7;
MoveJ RelTool (starting_position, -55, -202.4, -19 \Rx:=3.9, \Ry:=-32.7, \Rz:=0), v200, z200, Tooldata_7;
MoveJ RelTool (starting_position, -54, -203, -15 \Rx:=4.3, \Ry:=-32.7, \Rz:=0), v200, z200, Tooldata_7;
MoveJ RelTool (starting_position, -54, -203.6, -10 \Rx:=4.6, \Ry:=-32.7, \Rz:=0), v200, z200, Tooldata_7;
MoveJ RelTool (starting_position, -52, -204.1, -6 \Rx:=5, \Ry:=-32.4, \Rz:=0), v200, z200, Tooldata_7;
MoveJ RelTool (starting_position, -50, -204.6, -1 \Rx:=5.4, \Ry:=-32.1, \Rz:=0), v200, z200, Tooldata_7;
MoveJ RelTool (starting_position, -47, -205.1, 4 \Rx:=5.7, \Ry:=-31.5, \Rz:=0), v200, z200, Tooldata_7;
MoveJ RelTool (starting_position, -44, -205.6, 9 \Rx:=5.8, \Ry:=-30.9, \Rz:=0), v200, z200, Tooldata_7;
MoveJ RelTool (starting_position, -40, -206, 14 \Rx:=6, \Ry:=-30.3, \Rz:=0), v200, z200, Tooldata_7;
MoveJ RelTool (starting_position, -35, -206.4, 19 \Rx:=6.1, \Ry:=-29.4, \Rz:=0), v200, z200, Tooldata_7;
MoveJ RelTool (starting_position, -29, -206.8, 24 \Rx:=6.2, \Ry:=-28.5, \Rz:=0), v200, z200, Tooldata_7;
MoveJ RelTool (starting_position, -22, -207.1, 29 \Rx:=6.3, \Ry:=-27.3, \Rz:=0), v200, z200, Tooldata_7;
MoveJ RelTool (starting_position, -15, -207.5, 34 \Rx:=6.3, \Ry:=-26.1, \Rz:=0), v200, z200, Tooldata_7;
MoveJ RelTool (starting_position, -6, -207.7, 38 \Rx:=6.3, \Ry:=-24.3, \Rz:=0), v200, z200, Tooldata_7;
MoveJ RelTool (starting_position, 4, -208, 43 \Rx:=6.3, \Ry:=-22.8, \Rz:=0), v200, z200, Tooldata_7;
MoveJ RelTool (starting_position, 14, -208.3, 48 \Rx:=6.2, \Ry:=-21, \Rz:=0), v200, z200, Tooldata_7;
MoveJ RelTool (starting_position, 25, -208.5, 52 \Rx:=6.2, \Ry:=-18.9, \Rz:=0), v200, z200, Tooldata_7;
MoveJ RelTool (starting_position, 37, -208.7, 56 \Rx:=6.1, \Ry:=-16.8, \Rz:=0), v200, z200, Tooldata_7;
MoveJ RelTool (starting_position, 50, -208.9, 60 \Rx:=6, \Ry:=-14.4, \Rz:=0), v200, z200, Tooldata_7;
MoveJ RelTool (starting_position, 64, -209, 63 \Rx:=6, \Ry:=-12.3, \Rz:=0), v200, z200, Tooldata_7;
MoveJ RelTool (starting_position, 78, -209.2, 65 \Rx:=6, \Ry:=-9.9, \Rz:=0), v200, z200, Tooldata_7;
MoveJ RelTool (starting_position, 92, -209.3, 68 \Rx:=6.1, \Ry:=-7.2, \Rz:=0), v200, z200, Tooldata_7;
MoveJ RelTool (starting_position, 107, -209.4, 69 \Rx:=6.1, \Ry:=-4.8, \Rz:=0), v200, z200, Tooldata_7;
MoveJ RelTool (starting_position, 122, -209.5, 70 \Rx:=6.2, \Ry:=-1.8, \Rz:=0), v200, z200, Tooldata_7;
MoveJ RelTool (starting_position, 138, -209.6, 70 \Rx:=6.3, \Ry:=0.9, \Rz:=0), v200, z200, Tooldata_7;
MoveJ RelTool (starting_position, 154, -209.7, 69 \Rx:=6.4, \Ry:=3.6, \Rz:=0), v200, z200, Tooldata_7;
MoveJ RelTool (starting_position, 170, -209.8, 68 \Rx:=6.6, \Ry:=6.3, \Rz:=0), v200, z200, Tooldata_7;
MoveJ RelTool (starting_position, 185, -209.8, 65 \Rx:=6.8, \Ry:=9.3, \Rz:=0), v200, z200, Tooldata_7;
MoveJ RelTool (starting_position, 201, -209.9, 62 \Rx:=7, \Ry:=11.7, \Rz:=0), v200, z200, Tooldata_7;
MoveJ RelTool (starting_position, 216, -209.9, 58 \Rx:=7.1, \Ry:=14.4, \Rz:=0), v200, z200, Tooldata_7;
MoveJ RelTool (starting_position, 230, -210, 53 \Rx:=7.3, \Ry:=17.1, \Rz:=0), v200, z200, Tooldata_7;
MoveJ RelTool (starting_position, 244, -210, 48 \Rx:=7.5, \Ry:=19.5, \Rz:=0), v200, z200, Tooldata_7;
MoveJ RelTool (starting_position, 258, -210, 41 \Rx:=7.6, \Ry:=21.9, \Rz:=0), v200, z200, Tooldata_7;
MoveJ RelTool (starting_position, 270, -210, 34 \Rx:=7.9, \Ry:=24, \Rz:=0), v200, z200, Tooldata_7;
MoveJ RelTool (starting_position, 282, -210, 26 \Rx:=8.1, \Ry:=26.1, \Rz:=0), v200, z200, Tooldata_7;
MoveJ RelTool (starting_position, 293, -210, 17 \Rx:=8.2, \Ry:=27.9, \Rz:=0), v200, z200, Tooldata_7;
MoveJ RelTool (starting_position, 304, -210, 8 \Rx:=8.2, \Ry:=29.7, \Rz:=0), v200, z200, Tooldata_7;
MoveJ RelTool (starting_position, 313, -210.1, -2 \Rx:=8.2, \Ry:=31.5, \Rz:=0), v200, z200, Tooldata_7;
MoveJ RelTool (starting_position, 321, -210.1, -12 \Rx:=8.1, \Ry:=33, \Rz:=0), v200, z200, Tooldata_7;
MoveJ RelTool (starting_position, 329, -210.2, -22 \Rx:=8.1, \Ry:=34.2, \Rz:=0), v200, z200, Tooldata_7;
MoveJ RelTool (starting_position, 334, -210.3, -33 \Rx:=7.9, \Ry:=35.4, \Rz:=0), v200, z200, Tooldata_7;
MoveJ RelTool (starting_position, 338, -210.3, -44 \Rx:=7.6, \Ry:=36, \Rz:=0), v200, z200, Tooldata_7;
MoveJ RelTool (starting_position, 341, -210.4, -55 \Rx:=7.4, \Ry:=36.3, \Rz:=0), v200, z200, Tooldata_7;
MoveJ RelTool (starting_position, 342, -210.5, -66 \Rx:=7, \Ry:=36.6, \Rz:=0), v200, z200, Tooldata_7;
MoveJ RelTool (starting_position, 342, -210.7, -77 \Rx:=6.6, \Ry:=36.6, \Rz:=0), v200, z200, Tooldata_7;
MoveJ RelTool (starting_position, 340, -210.8, -88 \Rx:=6.1, \Ry:=36.3, \Rz:=0), v200, z200, Tooldata_7;
MoveJ RelTool (starting_position, 337, -210.9, -99 \Rx:=5.6, \Ry:=35.7, \Rz:=0), v200, z200, Tooldata_7;
MoveJ RelTool (starting_position, 333, -211.1, -110 \Rx:=5, \Ry:=34.8, \Rz:=0), v200, z200, Tooldata_7;
MoveJ RelTool (starting_position, 327, -211.3, -120 \Rx:=4.4, \Ry:=33.9, \Rz:=0), v200, z200, Tooldata_7;
MoveJ RelTool (starting_position, 319, -211.5, -130 \Rx:=3.9, \Ry:=32.4, \Rz:=0), v200, z200, Tooldata_7;
MoveJ RelTool (starting_position, 311, -211.7, -139 \Rx:=3.2, \Ry:=30.9, \Rz:=0), v200, z200, Tooldata_7;
MoveJ RelTool (starting_position, 301, -211.9, -148 \Rx:=2.6, \Ry:=29.1, \Rz:=0), v200, z200, Tooldata_7;
MoveJ RelTool (starting_position, 291, -212.2, -157 \Rx:=2.1, \Ry:=27.3, \Rz:=0), v200, z200, Tooldata_7;
MoveJ RelTool (starting_position, 279, -212.5, -165 \Rx:=1.7, \Ry:=25.5, \Rz:=0), v200, z200, Tooldata_7;
MoveJ RelTool (starting_position, 267, -212.8, -172 \Rx:=1.1, \Ry:=23.4, \Rz:=0), v200, z200, Tooldata_7;
MoveJ RelTool (starting_position, 253, -213.2, -178 \Rx:=0.6, \Ry:=21, \Rz:=0), v200, z200, Tooldata_7;
MoveJ RelTool (starting_position, 239, -213.6, -183 \Rx:=0.2, \Ry:=18.3, \Rz:=0), v200, z200, Tooldata_7;
MoveJ RelTool (starting_position, 224, -214, -187 \Rx:=-0.2, \Ry:=15.6, \Rz:=0), v200, z200, Tooldata_7;
MoveJ RelTool (starting_position, 209, -214.4, -191 \Rx:=-0.5, \Ry:=12.9, \Rz:=0), v200, z200, Tooldata_7;
MoveJ RelTool (starting_position, 193, -214.8, -193 \Rx:=-1, \Ry:=10.2, \Rz:=0), v200, z200, Tooldata_7;
MoveJ RelTool (starting_position, 178, -215.3, -193 \Rx:=-1.3, \Ry:=7.5, \Rz:=0), v200, z200, Tooldata_7;
MoveJ RelTool (starting_position, 162, -215.9, -193 \Rx:=-1.7, \Ry:=4.8, \Rz:=0), v200, z200, Tooldata_7;
MoveJ RelTool (starting_position, 147, -216.4, -192 \Rx:=-2, \Ry:=2.1, \Rz:=0), v200, z200, Tooldata_7;
MoveJ RelTool (starting_position, 132, -217, -189 \Rx:=-2.3, \Ry:=-0.6, \Rz:=0), v200, z200, Tooldata_7;
MoveJ RelTool (starting_position, 117, -217.6, -185 \Rx:=-2.6, \Ry:=-3, \Rz:=0), v200, z200, Tooldata_7;
MoveJ RelTool (starting_position, 103, -218.2, -179 \Rx:=-2.8, \Ry:=-5.7, \Rz:=0), v200, z200, Tooldata_7;
MoveJ RelTool (starting_position, 88, -218.8, -173 \Rx:=-3.1, \Ry:=-8.1, \Rz:=0), v200, z200, Tooldata_7;
MoveJ RelTool (starting_position, 75, -219.5, -165 \Rx:=-3.3, \Ry:=-10.5, \Rz:=0), v200, z200, Tooldata_7;
MoveJ RelTool (starting_position, 62, -220.2, -156 \Rx:=-3.5, \Ry:=-12.6, \Rz:=0), v200, z200, Tooldata_7;
MoveJ RelTool (starting_position, 49, -220.9, -146 \Rx:=-3.7, \Ry:=-15, \Rz:=0), v200, z200, Tooldata_7;
MoveJ RelTool (starting_position, 38, -221.6, -136 \Rx:=-3.8, \Ry:=-17.1, \Rz:=0), v200, z200, Tooldata_7;
MoveJ RelTool (starting_position, 27, -222.4, -124 \Rx:=-3.9, \Ry:=-18.9, \Rz:=0), v200, z200, Tooldata_7;
MoveJ RelTool (starting_position, 17, -223.1, -112 \Rx:=-4, \Ry:=-20.7, \Rz:=0), v200, z200, Tooldata_7;
MoveJ RelTool (starting_position, 9, -223.8, -99 \Rx:=-4.1, \Ry:=-22.2, \Rz:=0), v200, z200, Tooldata_7;
MoveJ RelTool (starting_position, 2, -224.6, -86 \Rx:=-4.1, \Ry:=-23.1, \Rz:=0), v200, z200, Tooldata_7;
MoveJ RelTool (starting_position, -3, -225.4, -72 \Rx:=-4.1, \Ry:=-24, \Rz:=0), v200, z200, Tooldata_7;
MoveJ RelTool (starting_position, -8, -226.1, -58 \Rx:=-4.2, \Ry:=-24.9, \Rz:=0), v200, z200, Tooldata_7;
MoveJ RelTool (starting_position, -12, -226.9, -44 \Rx:=-4.1, \Ry:=-25.5, \Rz:=0), v200, z200, Tooldata_7;
MoveJ RelTool (starting_position, -14, -227.6, -29 \Rx:=-4, \Ry:=-26.1, \Rz:=0), v200, z200, Tooldata_7;
MoveJ RelTool (starting_position, -15, -228.3, -15 \Rx:=-3.8, \Ry:=-26.4, \Rz:=0), v200, z200, Tooldata_7;
MoveJ RelTool (starting_position, -15, -229.1, 0 \Rx:=-3.7, \Ry:=-26.1, \Rz:=0), v200, z200, Tooldata_7;
MoveJ RelTool (starting_position, -13, -229.8, 14 \Rx:=-3.5, \Ry:=-25.8, \Rz:=0), v200, z200, Tooldata_7;
MoveJ RelTool (starting_position, -11, -230.5, 28 \Rx:=-3.3, \Ry:=-25.5, \Rz:=0), v200, z200, Tooldata_7;
MoveJ RelTool (starting_position, -7, -231.1, 42 \Rx:=-3.1, \Ry:=-24.6, \Rz:=0), v200, z200, Tooldata_7;
MoveJ RelTool (starting_position, -1, -231.8, 56 \Rx:=-2.8, \Ry:=-23.7, \Rz:=0), v200, z200, Tooldata_7;
MoveJ RelTool (starting_position, 5, -232.4, 70 \Rx:=-2.5, \Ry:=-22.5, \Rz:=0), v200, z200, Tooldata_7;
MoveJ RelTool (starting_position, 13, -233, 83 \Rx:=-2.1, \Ry:=-21.3, \Rz:=0), v200, z200, Tooldata_7;
MoveJ RelTool (starting_position, 21, -233.6, 95 \Rx:=-1.7, \Ry:=-19.8, \Rz:=0), v200, z200, Tooldata_7;
MoveJ RelTool (starting_position, 30, -234.1, 107 \Rx:=-1.3, \Ry:=-18, \Rz:=0), v200, z200, Tooldata_7;
MoveJ RelTool (starting_position, 40, -234.6, 118 \Rx:=-0.8, \Ry:=-16.2, \Rz:=0), v200, z200, Tooldata_7;
MoveJ RelTool (starting_position, 51, -235.1, 128 \Rx:=-0.3, \Ry:=-14.4, \Rz:=0), v200, z200, Tooldata_7;
MoveJ RelTool (starting_position, 61, -235.6, 138 \Rx:=0.2, \Ry:=-12.6, \Rz:=0), v200, z200, Tooldata_7;
MoveJ RelTool (starting_position, 73, -236, 147 \Rx:=0.7, \Ry:=-10.5, \Rz:=0), v200, z200, Tooldata_7;
MoveJ RelTool (starting_position, 84, -236.4, 155 \Rx:=1.2, \Ry:=-8.7, \Rz:=0), v200, z200, Tooldata_7;
MoveJ RelTool (starting_position, 96, -236.8, 162 \Rx:=1.7, \Ry:=-6.6, \Rz:=0), v200, z200, Tooldata_7;
MoveJ RelTool (starting_position, 108, -237.1, 167 \Rx:=2.2, \Ry:=-4.5, \Rz:=0), v200, z200, Tooldata_7;
MoveJ RelTool (starting_position, 120, -237.5, 172 \Rx:=2.6, \Ry:=-2.4, \Rz:=0), v200, z200, Tooldata_7;
MoveJ RelTool (starting_position, 132, -237.7, 176 \Rx:=3.1, \Ry:=-0, \Rz:=0), v200, z200, Tooldata_7;
MoveJ RelTool (starting_position, 144, -238, 179 \Rx:=3.5, \Ry:=1.8, \Rz:=0), v200, z200, Tooldata_7;
MoveJ RelTool (starting_position, 156, -238.3, 181 \Rx:=3.8, \Ry:=3.9, \Rz:=0), v200, z200, Tooldata_7;
MoveJ RelTool (starting_position, 167, -238.5, 183 \Rx:=4.2, \Ry:=6, \Rz:=0), v200, z200, Tooldata_7;
MoveJ RelTool (starting_position, 179, -238.7, 183 \Rx:=4.5, \Ry:=8.1, \Rz:=0), v200, z200, Tooldata_7;
MoveJ RelTool (starting_position, 189, -238.9, 182 \Rx:=4.7, \Ry:=9.9, \Rz:=0), v200, z200, Tooldata_7;
MoveJ RelTool (starting_position, 200, -239, 181 \Rx:=4.9, \Ry:=11.7, \Rz:=0), v200, z200, Tooldata_7;
MoveJ RelTool (starting_position, 209, -239.2, 180 \Rx:=5.1, \Ry:=13.2, \Rz:=0), v200, z200, Tooldata_7;
MoveJ RelTool (starting_position, 219, -239.3, 177 \Rx:=5.3, \Ry:=15, \Rz:=0), v200, z200, Tooldata_7;
MoveJ RelTool (starting_position, 228, -239.4, 175 \Rx:=5.5, \Ry:=16.5, \Rz:=0), v200, z200, Tooldata_7;
MoveJ RelTool (starting_position, 236, -239.5, 172 \Rx:=5.7, \Ry:=18, \Rz:=0), v200, z200, Tooldata_7;
MoveJ RelTool (starting_position, 243, -239.6, 168 \Rx:=5.9, \Ry:=19.2, \Rz:=0), v200, z200, Tooldata_7;
MoveJ RelTool (starting_position, 250, -239.7, 165 \Rx:=6.1, \Ry:=20.4, \Rz:=0), v200, z200, Tooldata_7;
MoveJ RelTool (starting_position, 257, -239.8, 161 \Rx:=6.2, \Ry:=21.6, \Rz:=0), v200, z200, Tooldata_7;
MoveJ RelTool (starting_position, 262, -239.8, 157 \Rx:=6.3, \Ry:=22.5, \Rz:=0), v200, z200, Tooldata_7;
MoveJ RelTool (starting_position, 267, -239.9, 153 \Rx:=6.4, \Ry:=23.4, \Rz:=0), v200, z200, Tooldata_7;
MoveJ RelTool (starting_position, 271, -239.9, 149 \Rx:=6.5, \Ry:=24, \Rz:=0), v200, z200, Tooldata_7;
MoveJ RelTool (starting_position, 274, -240, 144 \Rx:=6.6, \Ry:=24.6, \Rz:=0), v200, z200, Tooldata_7;
MoveJ RelTool (starting_position, 276, -240, 140 \Rx:=6.6, \Ry:=25.2, \Rz:=0), v200, z200, Tooldata_7;
MoveJ RelTool (starting_position, 278, -240, 136 \Rx:=6.6, \Ry:=25.2, \Rz:=0), v200, z200, Tooldata_7;
MoveJ RelTool (starting_position, 279, -240, 133 \Rx:=6.6, \Ry:=25.2, \Rz:=0), v200, z200, Tooldata_7;
MoveJ RelTool (starting_position, 279, -240, 129 \Rx:=6.5, \Ry:=25.2, \Rz:=0), v200, z200, Tooldata_7;
MoveJ RelTool (starting_position, 279, -240, 126 \Rx:=6.4, \Ry:=25.2, \Rz:=0), v200, z200, Tooldata_7;
MoveJ RelTool (starting_position, 279, -240, 122 \Rx:=6.3, \Ry:=25.2, \Rz:=0), v200, z200, Tooldata_7;
MoveJ RelTool (starting_position, 278, -240, 119 \Rx:=6.2, \Ry:=25.2, \Rz:=0), v200, z200, Tooldata_7;
MoveJ RelTool (starting_position, 278, -240, 116 \Rx:=6, \Ry:=24.9, \Rz:=0), v200, z200, Tooldata_7;
MoveJ RelTool (starting_position, 277, -240, 113 \Rx:=5.9, \Ry:=24.9, \Rz:=0), v200, z200, Tooldata_7;
MoveJ RelTool (starting_position, 275, -240, 110 \Rx:=5.8, \Ry:=24.6, \Rz:=0), v200, z200, Tooldata_7;
MoveJ RelTool (starting_position, 274, -240, 108 \Rx:=5.7, \Ry:=24.3, \Rz:=0), v200, z200, Tooldata_7;
MoveJ RelTool (starting_position, 272, -240, 105 \Rx:=5.6, \Ry:=24, \Rz:=0), v200, z200, Tooldata_7;
MoveJ RelTool (starting_position, 271, -240, 102 \Rx:=5.5, \Ry:=23.7, \Rz:=0), v200, z200, Tooldata_7;
MoveJ RelTool (starting_position, 269, -240, 100 \Rx:=5.5, \Ry:=23.4, \Rz:=0), v200, z200, Tooldata_7;
MoveJ RelTool (starting_position, 267, -240, 98 \Rx:=5.5, \Ry:=23.1, \Rz:=0), v200, z200, Tooldata_7;
MoveJ RelTool (starting_position, 265, -240, 95 \Rx:=5.6, \Ry:=22.8, \Rz:=0), v200, z200, Tooldata_7;
MoveJ RelTool (starting_position, 263, -240, 93 \Rx:=5.6, \Ry:=22.5, \Rz:=0), v200, z200, Tooldata_7;
MoveJ RelTool (starting_position, 260, -240, 91 \Rx:=5.8, \Ry:=21.9, \Rz:=0), v200, z200, Tooldata_7;
MoveJ RelTool (starting_position, 258, -240, 89 \Rx:=5.9, \Ry:=21.3, \Rz:=0), v200, z200, Tooldata_7;
MoveJ RelTool (starting_position, 256, -240, 87 \Rx:=6.2, \Ry:=21, \Rz:=0), v200, z200, Tooldata_7;
MoveJ RelTool (starting_position, 253, -240, 84 \Rx:=6.5, \Ry:=20.7, \Rz:=0), v200, z200, Tooldata_7;
MoveJ RelTool (starting_position, 251, -240, 82 \Rx:=6.8, \Ry:=20.4, \Rz:=0), v200, z200, Tooldata_7;
MoveJ RelTool (starting_position, 249, -240, 80 \Rx:=7.2, \Ry:=20.1, \Rz:=0), v200, z200, Tooldata_7;
MoveJ RelTool (starting_position, 246, -240.1, 78 \Rx:=7.5, \Ry:=19.5, \Rz:=0), v200, z200, Tooldata_7;
MoveJ RelTool (starting_position, 243, -240.1, 76 \Rx:=7.9, \Ry:=18.9, \Rz:=0), v200, z200, Tooldata_7;
MoveJ RelTool (starting_position, 241, -240.2, 74 \Rx:=8.3, \Ry:=18.3, \Rz:=0), v200, z200, Tooldata_7;
MoveJ RelTool (starting_position, 238, -240.3, 72 \Rx:=8.7, \Ry:=18, \Rz:=0), v200, z200, Tooldata_7;
MoveJ RelTool (starting_position, 236, -240.3, 70 \Rx:=9.2, \Ry:=17.7, \Rz:=0), v200, z200, Tooldata_7;
MoveJ RelTool (starting_position, 234, -240.4, 68 \Rx:=9.6, \Ry:=17.4, \Rz:=0), v200, z200, Tooldata_7;
MoveJ RelTool (starting_position, 232, -240.5, 66 \Rx:=10, \Ry:=17.1, \Rz:=0), v200, z200, Tooldata_7;
MoveJ RelTool (starting_position, 230, -240.7, 65 \Rx:=10.4, \Ry:=16.5, \Rz:=0), v200, z200, Tooldata_7;
MoveJ RelTool (starting_position, 228, -240.8, 63 \Rx:=10.8, \Ry:=16.2, \Rz:=0), v200, z200, Tooldata_7;
MoveJ RelTool (starting_position, 227, -240.9, 61 \Rx:=11.2, \Ry:=15.9, \Rz:=0), v200, z200, Tooldata_7;
MoveJ RelTool (starting_position, 225, -241.1, 59 \Rx:=11.6, \Ry:=15.9, \Rz:=0), v200, z200, Tooldata_7;
MoveJ RelTool (starting_position, 224, -241.3, 58 \Rx:=12, \Ry:=15.6, \Rz:=0), v200, z200, Tooldata_7;
MoveJ RelTool (starting_position, 223, -241.5, 56 \Rx:=12.4, \Ry:=15.6, \Rz:=0), v200, z200, Tooldata_7;
MoveJ RelTool (starting_position, 223, -241.7, 55 \Rx:=12.7, \Ry:=15.3, \Rz:=0), v200, z200, Tooldata_7;
MoveJ RelTool (starting_position, 222, -241.9, 53 \Rx:=13, \Ry:=15.3, \Rz:=0), v200, z200, Tooldata_7;
MoveJ RelTool (starting_position, 222, -242.2, 52 \Rx:=13.3, \Ry:=15, \Rz:=0), v200, z200, Tooldata_7;
MoveJ RelTool (starting_position, 222, -242.5, 51 \Rx:=13.6, \Ry:=15, \Rz:=0), v200, z200, Tooldata_7;
MoveJ RelTool (starting_position, 222, -242.8, 50 \Rx:=13.9, \Ry:=15.3, \Rz:=0), v200, z200, Tooldata_7;
MoveJ RelTool (starting_position, 223, -243.2, 48 \Rx:=14.1, \Ry:=15.3, \Rz:=0), v200, z200, Tooldata_7;
MoveJ RelTool (starting_position, 224, -243.6, 47 \Rx:=14.3, \Ry:=15.6, \Rz:=0), v200, z200, Tooldata_7;
MoveJ RelTool (starting_position, 225, -244, 46 \Rx:=14.5, \Ry:=15.9, \Rz:=0), v200, z200, Tooldata_7;
MoveJ RelTool (starting_position, 226, -244.4, 45 \Rx:=14.7, \Ry:=15.9, \Rz:=0), v200, z200, Tooldata_7;
MoveJ RelTool (starting_position, 228, -244.8, 44 \Rx:=14.9, \Ry:=16.2, \Rz:=0), v200, z200, Tooldata_7;
MoveJ RelTool (starting_position, 229, -245.3, 42 \Rx:=15, \Ry:=16.5, \Rz:=0), v200, z200, Tooldata_7;
MoveJ RelTool (starting_position, 231, -245.9, 41 \Rx:=15, \Ry:=16.8, \Rz:=0), v200, z200, Tooldata_7;
MoveJ RelTool (starting_position, 232, -246.4, 40 \Rx:=15, \Ry:=17.1, \Rz:=0), v200, z200, Tooldata_7;
MoveJ RelTool (starting_position, 234, -247, 38 \Rx:=15, \Ry:=17.4, \Rz:=0), v200, z200, Tooldata_7;
MoveJ RelTool (starting_position, 236, -247.6, 37 \Rx:=14.9, \Ry:=17.7, \Rz:=0), v200, z200, Tooldata_7;
MoveJ RelTool (starting_position, 238, -248.2, 35 \Rx:=14.8, \Ry:=18, \Rz:=0), v200, z200, Tooldata_7;
MoveJ RelTool (starting_position, 239, -248.8, 33 \Rx:=14.6, \Ry:=18.3, \Rz:=0), v200, z200, Tooldata_7;
MoveJ RelTool (starting_position, 241, -249.5, 31 \Rx:=14.4, \Ry:=18.6, \Rz:=0), v200, z200, Tooldata_7;
MoveJ RelTool (starting_position, 244, -250.2, 29 \Rx:=14.2, \Ry:=18.9, \Rz:=0), v200, z200, Tooldata_7;
MoveJ RelTool (starting_position, 246, -250.9, 27 \Rx:=13.9, \Ry:=19.5, \Rz:=0), v200, z200, Tooldata_7;
MoveJ RelTool (starting_position, 248, -251.6, 24 \Rx:=13.5, \Ry:=19.8, \Rz:=0), v200, z200, Tooldata_7;
MoveJ RelTool (starting_position, 251, -252.4, 21 \Rx:=13.1, \Ry:=20.4, \Rz:=0), v200, z200, Tooldata_7;
MoveJ RelTool (starting_position, 253, -253.1, 19 \Rx:=12.6, \Ry:=20.7, \Rz:=0), v200, z200, Tooldata_7;
MoveJ RelTool (starting_position, 256, -253.8, 16 \Rx:=12, \Ry:=21.3, \Rz:=0), v200, z200, Tooldata_7;
MoveJ RelTool (starting_position, 258, -254.6, 13 \Rx:=11.4, \Ry:=21.6, \Rz:=0), v200, z200, Tooldata_7;
MoveJ RelTool (starting_position, 260, -255.4, 10 \Rx:=10.6, \Ry:=21.9, \Rz:=0), v200, z200, Tooldata_7;
MoveJ RelTool (starting_position, 262, -256.1, 7 \Rx:=9.9, \Ry:=22.2, \Rz:=0), v200, z200, Tooldata_7;
MoveJ RelTool (starting_position, 263, -256.9, 4 \Rx:=9, \Ry:=22.5, \Rz:=0), v200, z200, Tooldata_7;
MoveJ RelTool (starting_position, 265, -257.6, 1 \Rx:=8.1, \Ry:=22.8, \Rz:=0), v200, z200, Tooldata_7;
MoveJ RelTool (starting_position, 266, -258.3, -2 \Rx:=7.2, \Ry:=23.1, \Rz:=0), v200, z200, Tooldata_7;
MoveJ RelTool (starting_position, 267, -259.1, -6 \Rx:=6.3, \Ry:=23.1, \Rz:=0), v200, z200, Tooldata_7;
MoveJ RelTool (starting_position, 267, -259.8, -9 \Rx:=5.3, \Ry:=23.1, \Rz:=0), v200, z200, Tooldata_7;
MoveJ RelTool (starting_position, 268, -260.5, -12 \Rx:=4.3, \Ry:=23.4, \Rz:=0), v200, z200, Tooldata_7;
MoveJ RelTool (starting_position, 268, -261.1, -15 \Rx:=3.3, \Ry:=23.4, \Rz:=0), v200, z200, Tooldata_7;
MoveJ RelTool (starting_position, 268, -261.8, -18 \Rx:=2.3, \Ry:=23.4, \Rz:=0), v200, z200, Tooldata_7;
MoveJ RelTool (starting_position, 268, -262.4, -22 \Rx:=1.3, \Ry:=23.1, \Rz:=0), v200, z200, Tooldata_7;
MoveJ RelTool (starting_position, 267, -263, -25 \Rx:=0.4, \Ry:=23.1, \Rz:=0), v200, z200, Tooldata_7;
MoveJ RelTool (starting_position, 266, -263.6, -28 \Rx:=-0.6, \Ry:=23.1, \Rz:=0), v200, z200, Tooldata_7;
MoveJ RelTool (starting_position, 265, -264.1, -31 \Rx:=-1.4, \Ry:=22.8, \Rz:=0), v200, z200, Tooldata_7;
MoveJ RelTool (starting_position, 264, -264.6, -34 \Rx:=-2.2, \Ry:=22.5, \Rz:=0), v200, z200, Tooldata_7;
MoveJ RelTool (starting_position, 262, -265.1, -36 \Rx:=-3, \Ry:=22.2, \Rz:=0), v200, z200, Tooldata_7;
MoveJ RelTool (starting_position, 261, -265.6, -39 \Rx:=-3.6, \Ry:=22.2, \Rz:=0), v200, z200, Tooldata_7;
MoveJ RelTool (starting_position, 259, -266, -42 \Rx:=-4.1, \Ry:=21.9, \Rz:=0), v200, z200, Tooldata_7;
MoveJ RelTool (starting_position, 257, -266.4, -45 \Rx:=-4.6, \Ry:=21.3, \Rz:=0), v200, z200, Tooldata_7;
MoveJ RelTool (starting_position, 255, -266.8, -47 \Rx:=-5.1, \Ry:=21, \Rz:=0), v200, z200, Tooldata_7;
MoveJ RelTool (starting_position, 253, -267.1, -50 \Rx:=-5.4, \Ry:=20.7, \Rz:=0), v200, z200, Tooldata_7;
MoveJ RelTool (starting_position, 251, -267.5, -52 \Rx:=-5.7, \Ry:=20.4, \Rz:=0), v200, z200, Tooldata_7;
MoveJ RelTool (starting_position, 249, -267.7, -54 \Rx:=-6, \Ry:=19.8, \Rz:=0), v200, z200, Tooldata_7;
MoveJ RelTool (starting_position, 247, -268, -56 \Rx:=-6.2, \Ry:=19.5, \Rz:=0), v200, z200, Tooldata_7;
MoveJ RelTool (starting_position, 244, -268.3, -58 \Rx:=-6.3, \Ry:=19.2, \Rz:=0), v200, z200, Tooldata_7;
MoveJ RelTool (starting_position, 242, -268.5, -60 \Rx:=-6.4, \Ry:=18.9, \Rz:=0), v200, z200, Tooldata_7;
MoveJ RelTool (starting_position, 239, -268.7, -62 \Rx:=-6.4, \Ry:=18.3, \Rz:=0), v200, z200, Tooldata_7;
MoveJ RelTool (starting_position, 237, -268.9, -64 \Rx:=-6.4, \Ry:=17.7, \Rz:=0), v200, z200, Tooldata_7;
MoveJ RelTool (starting_position, 234, -269, -65 \Rx:=-6.3, \Ry:=17.4, \Rz:=0), v200, z200, Tooldata_7;
MoveJ RelTool (starting_position, 231, -269.2, -67 \Rx:=-6.3, \Ry:=16.8, \Rz:=0), v200, z200, Tooldata_7;
MoveJ RelTool (starting_position, 229, -269.3, -68 \Rx:=-6.2, \Ry:=16.5, \Rz:=0), v200, z200, Tooldata_7;
MoveJ RelTool (starting_position, 226, -269.4, -70 \Rx:=-6.1, \Ry:=15.9, \Rz:=0), v200, z200, Tooldata_7;
MoveJ RelTool (starting_position, 223, -269.5, -71 \Rx:=-6, \Ry:=15.6, \Rz:=0), v200, z200, Tooldata_7;
MoveJ RelTool (starting_position, 220, -269.6, -73 \Rx:=-6, \Ry:=14.7, \Rz:=0), v200, z200, Tooldata_7;
MoveJ RelTool (starting_position, 217, -269.7, -74 \Rx:=-5.9, \Ry:=14.4, \Rz:=0), v200, z200, Tooldata_7;
MoveJ RelTool (starting_position, 214, -269.8, -75 \Rx:=-5.9, \Ry:=13.8, \Rz:=0), v200, z200, Tooldata_7;
MoveJ RelTool (starting_position, 212, -269.8, -77 \Rx:=-5.8, \Ry:=13.5, \Rz:=0), v200, z200, Tooldata_7;
MoveJ RelTool (starting_position, 210, -269.9, -78 \Rx:=-5.8, \Ry:=13.2, \Rz:=0), v200, z200, Tooldata_7;
MoveJ RelTool (starting_position, 207, -269.9, -79 \Rx:=-5.8, \Ry:=12.6, \Rz:=0), v200, z200, Tooldata_7;
MoveJ RelTool (starting_position, 205, -270, -80 \Rx:=-5.7, \Ry:=12.3, \Rz:=0), v200, z200, Tooldata_7;
MoveJ RelTool (starting_position, 203, -270, -81 \Rx:=-5.6, \Ry:=12, \Rz:=0), v200, z200, Tooldata_7;
MoveJ RelTool (starting_position, 201, -270, -83 \Rx:=-5.5, \Ry:=11.7, \Rz:=0), v200, z200, Tooldata_7;
MoveJ RelTool (starting_position, 200, -270, -84 \Rx:=-5.5, \Ry:=11.4, \Rz:=0), v200, z200, Tooldata_7;
MoveJ RelTool (starting_position, 198, -270, -85 \Rx:=-5.3, \Ry:=11.1, \Rz:=0), v200, z200, Tooldata_7;
MoveJ RelTool (starting_position, 196, -270, -86 \Rx:=-5.2, \Ry:=10.8, \Rz:=0), v200, z200, Tooldata_7;
MoveJ RelTool (starting_position, 194, -270, -87 \Rx:=-5, \Ry:=10.5, \Rz:=0), v200, z200, Tooldata_7;
MoveJ RelTool (starting_position, 193, -270, -88 \Rx:=-4.8, \Ry:=10.2, \Rz:=0), v200, z200, Tooldata_7;
MoveJ RelTool (starting_position, 191, -270, -89 \Rx:=-4.6, \Ry:=9.9, \Rz:=0), v200, z200, Tooldata_7;
MoveJ RelTool (starting_position, 189, -270, -90 \Rx:=-4.3, \Ry:=9.6, \Rz:=0), v200, z200, Tooldata_7;
MoveJ RelTool (starting_position, 188, -270, -91 \Rx:=-4, \Ry:=9.3, \Rz:=0), v200, z200, Tooldata_7;
MoveJ RelTool (starting_position, 186, -270, -92 \Rx:=-3.7, \Ry:=9, \Rz:=0), v200, z200, Tooldata_7;
MoveJ RelTool (starting_position, 185, -270, -93 \Rx:=-3.4, \Ry:=8.7, \Rz:=0), v200, z200, Tooldata_7;
MoveJ RelTool (starting_position, 183, -270, -94 \Rx:=-3, \Ry:=8.7, \Rz:=0), v200, z200, Tooldata_7;
MoveJ RelTool (starting_position, 182, -270, -94 \Rx:=-2.6, \Ry:=8.4, \Rz:=0), v200, z200, Tooldata_7;
MoveJ RelTool (starting_position, 181, -270, -95 \Rx:=-2.2, \Ry:=8.1, \Rz:=0), v200, z200, Tooldata_7;
MoveJ RelTool (starting_position, 180, -270, -96 \Rx:=-1.8, \Ry:=7.8, \Rz:=0), v200, z200, Tooldata_7;
MoveJ RelTool (starting_position, 179, -270, -97 \Rx:=-1.4, \Ry:=7.8, \Rz:=0), v200, z200, Tooldata_7;
MoveJ RelTool (starting_position, 178, -270, -98 \Rx:=-1.1, \Ry:=7.8, \Rz:=0), v200, z200, Tooldata_7;
MoveJ RelTool (starting_position, 177, -270, -98 \Rx:=-0.8, \Ry:=7.5, \Rz:=0), v200, z200, Tooldata_7;
MoveJ RelTool (starting_position, 176, -270, -99 \Rx:=-0.5, \Ry:=7.2, \Rz:=0), v200, z200, Tooldata_7;
MoveJ RelTool (starting_position, 175, -270, -100 \Rx:=-0.3, \Ry:=7.2, \Rz:=0), v200, z200, Tooldata_7;
MoveJ RelTool (starting_position, 174, -270, -100 \Rx:=-0.1, \Ry:=6.9, \Rz:=0), v200, z200, Tooldata_7;
MoveJ RelTool (starting_position, 173, -270, -101 \Rx:=0.1, \Ry:=6.9, \Rz:=0), v200, z200, Tooldata_7;
MoveJ RelTool (starting_position, 173, -270, -102 \Rx:=0.3, \Ry:=6.6, \Rz:=0), v200, z200, Tooldata_7;
MoveJ RelTool (starting_position, 172, -270, -102 \Rx:=0.5, \Ry:=6.6, \Rz:=0), v200, z200, Tooldata_7;
MoveJ RelTool (starting_position, 172, -270, -103 \Rx:=0.7, \Ry:=6.6, \Rz:=0), v200, z200, Tooldata_7;
MoveJ RelTool (starting_position, 172, -270, -103 \Rx:=0.7, \Ry:=6.6, \Rz:=0), v200, z200, Tooldata_7;
MoveJ RelTool (starting_position, 172, -270, -104 \Rx:=0.8, \Ry:=6.6, \Rz:=0), v200, z200, Tooldata_7;
MoveJ RelTool (starting_position, 172, -270, -104 \Rx:=0.9, \Ry:=6.6, \Rz:=0), v200, z200, Tooldata_7;
MoveJ RelTool (starting_position, 171, -270, -105 \Rx:=1, \Ry:=6.6, \Rz:=0), v200, z200, Tooldata_7;
MoveJ RelTool (starting_position, 171, -270, -106 \Rx:=1.1, \Ry:=6.6, \Rz:=0), v200, z200, Tooldata_7;
MoveJ RelTool (starting_position, 170, -270, -106 \Rx:=1.1, \Ry:=6.3, \Rz:=0), v200, z200, Tooldata_7;
MoveJ RelTool (starting_position, 170, -270, -107 \Rx:=1.2, \Ry:=6.3, \Rz:=0), v200, z200, Tooldata_7;
MoveJ RelTool (starting_position, 169, -270, -108 \Rx:=1.3, \Ry:=6, \Rz:=0), v200, z200, Tooldata_7;
MoveJ RelTool (starting_position, 168, -270, -108 \Rx:=1.4, \Ry:=6, \Rz:=0), v200, z200, Tooldata_7;
MoveJ RelTool (starting_position, 167, -270, -109 \Rx:=1.4, \Ry:=5.7, \Rz:=0), v200, z200, Tooldata_7;
MoveJ RelTool (starting_position, 167, -270, -110 \Rx:=1.5, \Ry:=5.7, \Rz:=0), v200, z200, Tooldata_7;
MoveJ RelTool (starting_position, 166, -270, -110 \Rx:=1.5, \Ry:=5.7, \Rz:=0), v200, z200, Tooldata_7;
MoveJ RelTool (starting_position, 166, -270, -111 \Rx:=1.4, \Ry:=5.4, \Rz:=0), v200, z200, Tooldata_7;
MoveJ RelTool (starting_position, 165, -270, -112 \Rx:=1.4, \Ry:=5.4, \Rz:=0), v200, z200, Tooldata_7;
MoveJ RelTool (starting_position, 164, -270, -113 \Rx:=1.3, \Ry:=5.4, \Rz:=0), v200, z200, Tooldata_7;
MoveJ RelTool (starting_position, 164, -270, -113 \Rx:=1.3, \Ry:=5.1, \Rz:=0), v200, z200, Tooldata_7;
MoveJ RelTool (starting_position, 163, -270, -114 \Rx:=1.2, \Ry:=5.1, \Rz:=0), v200, z200, Tooldata_7;
MoveJ RelTool (starting_position, 162, -270, -115 \Rx:=1.2, \Ry:=5.1, \Rz:=0), v200, z200, Tooldata_7;
MoveJ RelTool (starting_position, 162, -270, -116 \Rx:=1.1, \Ry:=4.8, \Rz:=0), v200, z200, Tooldata_7;
MoveJ RelTool (starting_position, 161, -270, -116 \Rx:=1.1, \Ry:=4.8, \Rz:=0), v200, z200, Tooldata_7;
MoveJ RelTool (starting_position, 160, -270, -117 \Rx:=1, \Ry:=4.5, \Rz:=0), v200, z200, Tooldata_7;
MoveJ RelTool (starting_position, 159, -270, -118 \Rx:=0.9, \Ry:=4.2, \Rz:=0), v200, z200, Tooldata_7;
MoveJ RelTool (starting_position, 157, -270, -118 \Rx:=0.8, \Ry:=4.2, \Rz:=0), v200, z200, Tooldata_7;
MoveJ RelTool (starting_position, 156, -270, -119 \Rx:=0.6, \Ry:=3.9, \Rz:=0), v200, z200, Tooldata_7;
MoveJ RelTool (starting_position, 155, -270, -120 \Rx:=0.4, \Ry:=3.6, \Rz:=0), v200, z200, Tooldata_7;
MoveJ RelTool (starting_position, 154, -270, -120 \Rx:=0.2, \Ry:=3.6, \Rz:=0), v200, z200, Tooldata_7;
MoveJ RelTool (starting_position, 153, -270, -121 \Rx:=-0, \Ry:=3.3, \Rz:=0), v200, z200, Tooldata_7;
MoveJ RelTool (starting_position, 151, -270, -121 \Rx:=-0.2, \Ry:=3, \Rz:=0), v200, z200, Tooldata_7;
MoveJ RelTool (starting_position, 150, -270, -121 \Rx:=-0.5, \Ry:=2.7, \Rz:=0), v200, z200, Tooldata_7;
MoveJ RelTool (starting_position, 148, -270, -122 \Rx:=-0.7, \Ry:=2.4, \Rz:=0), v200, z200, Tooldata_7;
MoveJ RelTool (starting_position, 147, -270, -122 \Rx:=-1, \Ry:=2.4, \Rz:=0), v200, z200, Tooldata_7;
MoveJ RelTool (starting_position, 146, -270, -122 \Rx:=-1.4, \Ry:=2.1, \Rz:=0), v200, z200, Tooldata_7;
MoveJ RelTool (starting_position, 144, -270, -123 \Rx:=-1.6, \Ry:=1.8, \Rz:=0), v200, z200, Tooldata_7;
MoveJ RelTool (starting_position, 143, -270, -123 \Rx:=-2, \Ry:=1.5, \Rz:=0), v200, z200, Tooldata_7;
MoveJ RelTool (starting_position, 141, -270, -123 \Rx:=-2.4, \Ry:=1.2, \Rz:=0), v200, z200, Tooldata_7;
MoveJ RelTool (starting_position, 140, -270, -123 \Rx:=-2.8, \Ry:=0.9, \Rz:=0), v200, z200, Tooldata_7;
MoveJ RelTool (starting_position, 138, -270, -123 \Rx:=-3.3, \Ry:=0.9, \Rz:=0), v200, z200, Tooldata_7;
MoveJ RelTool (starting_position, 137, -270, -123 \Rx:=-3.7, \Ry:=0.6, \Rz:=0), v200, z200, Tooldata_7;
MoveJ RelTool (starting_position, 136, -270, -123 \Rx:=-4.2, \Ry:=0.3, \Rz:=0), v200, z200, Tooldata_7;
MoveJ RelTool (starting_position, 135, -270.1, -122 \Rx:=-4.7, \Ry:=0.3, \Rz:=0), v200, z200, Tooldata_7;
MoveJ RelTool (starting_position, 135, -270.1, -122 \Rx:=-5.1, \Ry:=0, \Rz:=0), v200, z200, Tooldata_7;
MoveJ RelTool (starting_position, 134, -270.2, -122 \Rx:=-5.5, \Ry:=-0, \Rz:=0), v200, z200, Tooldata_7;
MoveJ RelTool (starting_position, 133, -270.3, -122 \Rx:=-5.8, \Ry:=-0, \Rz:=0), v200, z200, Tooldata_7;
MoveJ RelTool (starting_position, 133, -270.3, -121 \Rx:=-6.1, \Ry:=-0.3, \Rz:=0), v200, z200, Tooldata_7;
MoveJ RelTool (starting_position, 132, -270.4, -121 \Rx:=-6.3, \Ry:=-0.3, \Rz:=0), v200, z200, Tooldata_7;
MoveJ RelTool (starting_position, 132, -270.5, -120 \Rx:=-6.5, \Ry:=-0.3, \Rz:=0), v200, z200, Tooldata_7;
MoveJ RelTool (starting_position, 132, -270.7, -120 \Rx:=-6.7, \Ry:=-0.3, \Rz:=0), v200, z200, Tooldata_7;
MoveJ RelTool (starting_position, 132, -270.8, -120 \Rx:=-6.9, \Ry:=-0.3, \Rz:=0), v200, z200, Tooldata_7;
MoveJ RelTool (starting_position, 132, -270.9, -119 \Rx:=-7, \Ry:=-0.3, \Rz:=0), v200, z200, Tooldata_7;
MoveJ RelTool (starting_position, 132, -271.1, -119 \Rx:=-7.1, \Ry:=-0.3, \Rz:=0), v200, z200, Tooldata_7;
MoveJ RelTool (starting_position, 132, -271.3, -119 \Rx:=-7, \Ry:=-0.3, \Rz:=0), v200, z200, Tooldata_7;
MoveJ RelTool (starting_position, 132, -271.5, -118 \Rx:=-7, \Ry:=-0.3, \Rz:=0), v200, z200, Tooldata_7;
MoveJ RelTool (starting_position, 132, -271.7, -118 \Rx:=-6.8, \Ry:=-0.3, \Rz:=0), v200, z200, Tooldata_7;
MoveJ RelTool (starting_position, 132, -271.9, -118 \Rx:=-6.7, \Ry:=-0.3, \Rz:=0), v200, z200, Tooldata_7;
MoveJ RelTool (starting_position, 132, -272.2, -118 \Rx:=-6.4, \Ry:=-0.3, \Rz:=0), v200, z200, Tooldata_7;
MoveJ RelTool (starting_position, 132, -272.5, -118 \Rx:=-6.1, \Ry:=-0.3, \Rz:=0), v200, z200, Tooldata_7;
MoveJ RelTool (starting_position, 132, -272.8, -118 \Rx:=-5.8, \Ry:=-0.3, \Rz:=0), v200, z200, Tooldata_7;
MoveJ RelTool (starting_position, 133, -273.2, -118 \Rx:=-5.4, \Ry:=-0.3, \Rz:=0), v200, z200, Tooldata_7;
MoveJ RelTool (starting_position, 134, -273.6, -118 \Rx:=-5, \Ry:=-0, \Rz:=0), v200, z200, Tooldata_7;
MoveJ RelTool (starting_position, 134, -274, -118 \Rx:=-4.6, \Ry:=-0, \Rz:=0), v200, z200, Tooldata_7;
MoveJ RelTool (starting_position, 135, -274.4, -118 \Rx:=-4.1, \Ry:=0.3, \Rz:=0), v200, z200, Tooldata_7;
MoveJ RelTool (starting_position, 136, -274.8, -118 \Rx:=-3.6, \Ry:=0.6, \Rz:=0), v200, z200, Tooldata_7;
MoveJ RelTool (starting_position, 137, -275.3, -118 \Rx:=-3.1, \Ry:=0.6, \Rz:=0), v200, z200, Tooldata_7;
MoveJ RelTool (starting_position, 137, -275.9, -119 \Rx:=-2.6, \Ry:=0.6, \Rz:=0), v200, z200, Tooldata_7;
MoveJ RelTool (starting_position, 137, -276.4, -119 \Rx:=-2.2, \Ry:=0.6, \Rz:=0), v200, z200, Tooldata_7;
MoveJ RelTool (starting_position, 137, -277, -119 \Rx:=-1.7, \Ry:=0.6, \Rz:=0), v200, z200, Tooldata_7;
MoveJ RelTool (starting_position, 137, -277.6, -119 \Rx:=-1.3, \Ry:=0.6, \Rz:=0), v200, z200, Tooldata_7;
MoveJ RelTool (starting_position, 138, -278.2, -119 \Rx:=-1, \Ry:=0.6, \Rz:=0), v200, z200, Tooldata_7;
MoveJ RelTool (starting_position, 138, -278.8, -120 \Rx:=-0.7, \Ry:=0.6, \Rz:=0), v200, z200, Tooldata_7;
MoveJ RelTool (starting_position, 138, -279.5, -120 \Rx:=-0.4, \Ry:=0.9, \Rz:=0), v200, z200, Tooldata_7;
MoveJ RelTool (starting_position, 139, -280.2, -120 \Rx:=-0.1, \Ry:=0.9, \Rz:=0), v200, z200, Tooldata_7;
MoveJ RelTool (starting_position, 139, -280.9, -120 \Rx:=0, \Ry:=0.9, \Rz:=0), v200, z200, Tooldata_7;
MoveJ RelTool (starting_position, 139, -281.6, -120 \Rx:=0.2, \Ry:=0.9, \Rz:=0), v200, z200, Tooldata_7;
MoveJ RelTool (starting_position, 140, -282.4, -120 \Rx:=0.3, \Ry:=0.9, \Rz:=0), v200, z200, Tooldata_7;
MoveJ RelTool (starting_position, 140, -283.1, -120 \Rx:=0.4, \Ry:=1.2, \Rz:=0), v200, z200, Tooldata_7;
MoveJ RelTool (starting_position, 140, -283.8, -120 \Rx:=0.4, \Ry:=1.2, \Rz:=0), v200, z200, Tooldata_7;
MoveJ RelTool (starting_position, 140, -284.6, -121 \Rx:=0.5, \Ry:=1.2, \Rz:=0), v200, z200, Tooldata_7;
MoveJ RelTool (starting_position, 141, -285.4, -121 \Rx:=0.4, \Ry:=1.2, \Rz:=0), v200, z200, Tooldata_7;
MoveJ RelTool (starting_position, 141, -286.1, -121 \Rx:=0.4, \Ry:=1.2, \Rz:=0), v200, z200, Tooldata_7;
MoveJ RelTool (starting_position, 141, -286.9, -121 \Rx:=0.4, \Ry:=1.2, \Rz:=0), v200, z200, Tooldata_7;
MoveJ RelTool (starting_position, 141, -287.6, -121 \Rx:=0.4, \Ry:=1.2, \Rz:=0), v200, z200, Tooldata_7;
MoveJ RelTool (starting_position, 141, -288.3, -121 \Rx:=0.3, \Ry:=1.2, \Rz:=0), v200, z200, Tooldata_7;
MoveJ RelTool (starting_position, 141, -289.1, -121 \Rx:=0.2, \Ry:=1.2, \Rz:=0), v200, z200, Tooldata_7;
MoveJ RelTool (starting_position, 141, -289.8, -121 \Rx:=0.2, \Ry:=1.2, \Rz:=0), v200, z200, Tooldata_7;
MoveJ RelTool (starting_position, 141, -290.5, -121 \Rx:=0.1, \Ry:=1.2, \Rz:=0), v200, z200, Tooldata_7;
MoveJ RelTool (starting_position, 142, -291.1, -121 \Rx:=0.1, \Ry:=1.2, \Rz:=0), v200, z200, Tooldata_7;
MoveJ RelTool (starting_position, 142, -291.8, -121 \Rx:=0.1, \Ry:=1.5, \Rz:=0), v200, z200, Tooldata_7;
MoveJ RelTool (starting_position, 143, -292.4, -121 \Rx:=0.1, \Ry:=1.5, \Rz:=0), v200, z200, Tooldata_7;
MoveJ RelTool (starting_position, 143, -293, -121 \Rx:=0.2, \Ry:=1.8, \Rz:=0), v200, z200, Tooldata_7;
MoveJ RelTool (starting_position, 144, -293.6, -121 \Rx:=0.2, \Ry:=1.8, \Rz:=0), v200, z200, Tooldata_7;
MoveJ RelTool (starting_position, 144, -294.1, -120 \Rx:=0.3, \Ry:=1.8, \Rz:=0), v200, z200, Tooldata_7;
MoveJ RelTool (starting_position, 144, -294.6, -120 \Rx:=0.4, \Ry:=1.8, \Rz:=0), v200, z200, Tooldata_7;
MoveJ RelTool (starting_position, 144, -295.1, -120 \Rx:=0.6, \Ry:=1.8, \Rz:=0), v200, z200, Tooldata_7;
MoveJ RelTool (starting_position, 144, -295.6, -120 \Rx:=0.7, \Ry:=1.8, \Rz:=0), v200, z200, Tooldata_7;
MoveJ RelTool (starting_position, 145, -296, -120 \Rx:=0.9, \Ry:=1.8, \Rz:=0), v200, z200, Tooldata_7;
MoveJ RelTool (starting_position, 145, -296.4, -120 \Rx:=1.1, \Ry:=1.8, \Rz:=0), v200, z200, Tooldata_7;
MoveJ RelTool (starting_position, 145, -296.8, -119 \Rx:=1.4, \Ry:=2.1, \Rz:=0), v200, z200, Tooldata_7;
MoveJ RelTool (starting_position, 146, -297.1, -119 \Rx:=1.6, \Ry:=2.1, \Rz:=0), v200, z200, Tooldata_7;
MoveJ RelTool (starting_position, 146, -297.5, -119 \Rx:=1.9, \Ry:=2.1, \Rz:=0), v200, z200, Tooldata_7;
MoveJ RelTool (starting_position, 147, -297.7, -118 \Rx:=2.1, \Ry:=2.4, \Rz:=0), v200, z200, Tooldata_7;
MoveJ RelTool (starting_position, 147, -298, -118 \Rx:=2.3, \Ry:=2.4, \Rz:=0), v200, z200, Tooldata_7;
MoveJ RelTool (starting_position, 147, -298.3, -118 \Rx:=2.5, \Ry:=2.4, \Rz:=0), v200, z200, Tooldata_7;
MoveJ RelTool (starting_position, 148, -298.5, -117 \Rx:=2.6, \Ry:=2.4, \Rz:=0), v200, z200, Tooldata_7;
MoveJ RelTool (starting_position, 148, -298.7, -117 \Rx:=2.7, \Ry:=2.4, \Rz:=0), v200, z200, Tooldata_7;
MoveJ RelTool (starting_position, 148, -298.9, -116 \Rx:=2.7, \Ry:=2.4, \Rz:=0), v200, z200, Tooldata_7;
MoveJ RelTool (starting_position, 149, -299, -116 \Rx:=2.7, \Ry:=2.7, \Rz:=0), v200, z200, Tooldata_7;
MoveJ RelTool (starting_position, 149, -299.2, -116 \Rx:=2.7, \Ry:=2.7, \Rz:=0), v200, z200, Tooldata_7;
MoveJ RelTool (starting_position, 149, -299.3, -115 \Rx:=2.7, \Ry:=2.7, \Rz:=0), v200, z200, Tooldata_7;
MoveJ RelTool (starting_position, 149, -299.4, -115 \Rx:=2.6, \Ry:=2.7, \Rz:=0), v200, z200, Tooldata_7;
MoveJ RelTool (starting_position, 149, -299.5, -115 \Rx:=2.5, \Ry:=2.7, \Rz:=0), v200, z200, Tooldata_7;
MoveJ RelTool (starting_position, 149, -299.6, -114 \Rx:=2.4, \Ry:=2.7, \Rz:=0), v200, z200, Tooldata_7;
MoveJ RelTool (starting_position, 149, -299.7, -114 \Rx:=2.2, \Ry:=2.7, \Rz:=0), v200, z200, Tooldata_7;
MoveJ RelTool (starting_position, 149, -299.8, -114 \Rx:=2, \Ry:=2.7, \Rz:=0), v200, z200, Tooldata_7;
MoveJ RelTool (starting_position, 149, -299.8, -114 \Rx:=1.8, \Ry:=2.7, \Rz:=0), v200, z200, Tooldata_7;
MoveJ RelTool (starting_position, 149, -299.9, -113 \Rx:=1.7, \Ry:=2.7, \Rz:=0), v200, z200, Tooldata_7;
MoveJ RelTool (starting_position, 149, -299.9, -113 \Rx:=1.5, \Ry:=2.7, \Rz:=0), v200, z200, Tooldata_7;
MoveJ RelTool (starting_position, 149, -300, -113 \Rx:=1.3, \Ry:=2.7, \Rz:=0), v200, z200, Tooldata_7;
MoveJ RelTool (starting_position, 149, -300, -113 \Rx:=1.1, \Ry:=2.7, \Rz:=0), v200, z200, Tooldata_7;
MoveJ RelTool (starting_position, 148, -300, -113 \Rx:=1, \Ry:=2.4, \Rz:=0), v200, z200, Tooldata_7;
MoveJ RelTool (starting_position, 148, -300, -113 \Rx:=0.9, \Ry:=2.4, \Rz:=0), v200, z200, Tooldata_7;
MoveJ RelTool (starting_position, 147, -300, -113 \Rx:=0.7, \Ry:=2.4, \Rz:=0), v200, z200, Tooldata_7;
MoveJ RelTool (starting_position, 147, -300, -113 \Rx:=0.6, \Ry:=2.4, \Rz:=0), v200, z200, Tooldata_7;
MoveJ RelTool (starting_position, 146, -300, -113 \Rx:=0.5, \Ry:=2.1, \Rz:=0), v200, z200, Tooldata_7;
MoveJ RelTool (starting_position, 146, -300, -113 \Rx:=0.4, \Ry:=2.1, \Rz:=0), v200, z200, Tooldata_7;
MoveJ RelTool (starting_position, 145, -300, -113 \Rx:=0.2, \Ry:=2.1, \Rz:=0), v200, z200, Tooldata_7;
MoveJ RelTool (starting_position, 144, -300, -113 \Rx:=0.1, \Ry:=1.8, \Rz:=0), v200, z200, Tooldata_7;
MoveJ RelTool (starting_position, 144, -300, -113 \Rx:=0.1, \Ry:=1.8, \Rz:=0), v200, z200, Tooldata_7;
MoveJ RelTool (starting_position, 143, -300, -114 \Rx:=-0, \Ry:=1.5, \Rz:=0), v200, z200, Tooldata_7;
MoveJ RelTool (starting_position, 142, -300, -114 \Rx:=-0.1, \Ry:=1.5, \Rz:=0), v200, z200, Tooldata_7;
MoveJ RelTool (starting_position, 141, -300, -114 \Rx:=-0.1, \Ry:=1.2, \Rz:=0), v200, z200, Tooldata_7;
MoveJ RelTool (starting_position, 140, -300, -114 \Rx:=-0.1, \Ry:=1.2, \Rz:=0), v200, z200, Tooldata_7;
MoveJ RelTool (starting_position, 140, -300, -114 \Rx:=-0.2, \Ry:=0.9, \Rz:=0), v200, z200, Tooldata_7;
MoveJ RelTool (starting_position, 139, -300, -114 \Rx:=-0.2, \Ry:=0.9, \Rz:=0), v200, z200, Tooldata_7;
MoveJ RelTool (starting_position, 138, -300, -115 \Rx:=-0.2, \Ry:=0.9, \Rz:=0), v200, z200, Tooldata_7;
MoveJ RelTool (starting_position, 138, -300, -115 \Rx:=-0.2, \Ry:=0.6, \Rz:=0), v200, z200, Tooldata_7;
MoveJ RelTool (starting_position, 137, -300, -115 \Rx:=-0.2, \Ry:=0.6, \Rz:=0), v200, z200, Tooldata_7;
MoveJ RelTool (starting_position, 136, -300, -115 \Rx:=-0.2, \Ry:=0.3, \Rz:=0), v200, z200, Tooldata_7;
MoveJ RelTool (starting_position, 135, -300, -115 \Rx:=-0.2, \Ry:=0.3, \Rz:=0), v200, z200, Tooldata_7;
MoveJ RelTool (starting_position, 135, -300, -115 \Rx:=-0.2, \Ry:=0.3, \Rz:=0), v200, z200, Tooldata_7;
MoveJ RelTool (starting_position, 134, -300, -115 \Rx:=-0.2, \Ry:=-0, \Rz:=0), v200, z200, Tooldata_7;
MoveJ RelTool (starting_position, 133, -300, -115 \Rx:=-0.2, \Ry:=-0.3, \Rz:=0), v200, z200, Tooldata_7;
MoveJ RelTool (starting_position, 132, -300, -116 \Rx:=-0.2, \Ry:=-0.3, \Rz:=0), v200, z200, Tooldata_7;
MoveJ RelTool (starting_position, 131, -300, -116 \Rx:=-0.2, \Ry:=-0.6, \Rz:=0), v200, z200, Tooldata_7;
MoveJ RelTool (starting_position, 131, -300, -116 \Rx:=-0.2, \Ry:=-0.6, \Rz:=0), v200, z200, Tooldata_7;
MoveJ RelTool (starting_position, 131, -300, -115 \Rx:=-0.2, \Ry:=-0.6, \Rz:=0), v200, z200, Tooldata_7;
MoveJ RelTool (starting_position, 131, -300, -115 \Rx:=-0.2, \Ry:=-0.3, \Rz:=0), v200, z200, Tooldata_7;
MoveJ RelTool (starting_position, 131, -300, -115 \Rx:=-0.2, \Ry:=-0.6, \Rz:=0), v200, z200, Tooldata_7;
MoveJ RelTool (starting_position, 130, -300, -115 \Rx:=-0.2, \Ry:=-0.6, \Rz:=0), v200, z200, Tooldata_7;
MoveJ RelTool (starting_position, 130, -300, -115 \Rx:=-0.3, \Ry:=-0.6, \Rz:=0), v200, z200, Tooldata_7;
MoveJ RelTool (starting_position, 130, -300, -115 \Rx:=-0.3, \Ry:=-0.6, \Rz:=0), v200, z200, Tooldata_7;
MoveJ RelTool (starting_position, 130, -300, -114 \Rx:=-0.4, \Ry:=-0.6, \Rz:=0), v200, z200, Tooldata_7;
MoveJ RelTool (starting_position, 130, -300, -114 \Rx:=-0.6, \Ry:=-0.6, \Rz:=0), v200, z200, Tooldata_7;
MoveJ RelTool (starting_position, 131, -300, -114 \Rx:=-0.7, \Ry:=-0.6, \Rz:=0), v200, z200, Tooldata_7;
MoveJ RelTool (starting_position, 131, -300, -113 \Rx:=-0.9, \Ry:=-0.6, \Rz:=0), v200, z200, Tooldata_7;
MoveJ RelTool (starting_position, 132, -300, -113 \Rx:=-1.1, \Ry:=-0.3, \Rz:=0), v200, z200, Tooldata_7;
MoveJ RelTool (starting_position, 133, -300, -112 \Rx:=-1.4, \Ry:=-0.3, \Rz:=0), v200, z200, Tooldata_7;
MoveJ RelTool (starting_position, 134, -300, -112 \Rx:=-1.7, \Ry:=0, \Rz:=0), v200, z200, Tooldata_7;
MoveJ RelTool (starting_position, 136, -300, -112 \Rx:=-2.1, \Ry:=0.3, \Rz:=0), v200, z200, Tooldata_7;
MoveJ RelTool (starting_position, 137, -300, -111 \Rx:=-2.5, \Ry:=0.6, \Rz:=0), v200, z200, Tooldata_7;
MoveJ RelTool (starting_position, 139, -300, -111 \Rx:=-2.9, \Ry:=0.9, \Rz:=0), v200, z200, Tooldata_7;
MoveJ RelTool (starting_position, 141, -300, -111 \Rx:=-3.4, \Ry:=1.2, \Rz:=0), v200, z200, Tooldata_7;
MoveJ RelTool (starting_position, 144, -300, -110 \Rx:=-3.9, \Ry:=1.8, \Rz:=0), v200, z200, Tooldata_7;
MoveJ RelTool (starting_position, 147, -300, -110 \Rx:=-4.5, \Ry:=2.1, \Rz:=0), v200, z200, Tooldata_7;
MoveJ RelTool (starting_position, 149, -300, -110 \Rx:=-5.1, \Ry:=2.7, \Rz:=0), v200, z200, Tooldata_7;
MoveJ RelTool (starting_position, 152, -300, -110 \Rx:=-5.8, \Ry:=3.3, \Rz:=0), v200, z200, Tooldata_7;
MoveJ RelTool (starting_position, 155, -300, -110 \Rx:=-6.4, \Ry:=3.6, \Rz:=0), v200, z200, Tooldata_7;
MoveJ RelTool (starting_position, 158, -300, -110 \Rx:=-7.1, \Ry:=4.2, \Rz:=0), v200, z200, Tooldata_7;
MoveJ RelTool (starting_position, 161, -300, -111 \Rx:=-7.8, \Ry:=4.8, \Rz:=0), v200, z200, Tooldata_7;
MoveJ RelTool (starting_position, 164, -300, -111 \Rx:=-8.5, \Ry:=5.1, \Rz:=0), v200, z200, Tooldata_7;
MoveJ RelTool (starting_position, 167, -300, -112 \Rx:=-9.2, \Ry:=5.7, \Rz:=0), v200, z200, Tooldata_7;
MoveJ RelTool (starting_position, 170, -300, -112 \Rx:=-9.8, \Ry:=6.3, \Rz:=0), v200, z200, Tooldata_7;
MoveJ RelTool (starting_position, 173, -300, -113 \Rx:=-10.5, \Ry:=6.9, \Rz:=0), v200, z200, Tooldata_7;
MoveJ RelTool (starting_position, 176, -300, -114 \Rx:=-11.1, \Ry:=7.2, \Rz:=0), v200, z200, Tooldata_7;
MoveJ RelTool (starting_position, 179, -300, -115 \Rx:=-11.7, \Ry:=7.8, \Rz:=0), v200, z200, Tooldata_7;
MoveJ RelTool (starting_position, 182, -300, -116 \Rx:=-12.3, \Ry:=8.4, \Rz:=0), v200, z200, Tooldata_7;
MoveJ RelTool (starting_position, 184, -300, -117 \Rx:=-12.8, \Ry:=8.7, \Rz:=0), v200, z200, Tooldata_7;
MoveJ RelTool (starting_position, 187, -300, -118 \Rx:=-13.3, \Ry:=9.3, \Rz:=0), v200, z200, Tooldata_7;
MoveJ RelTool (starting_position, 190, -300, -119 \Rx:=-13.8, \Ry:=9.9, \Rz:=0), v200, z200, Tooldata_7;
MoveJ RelTool (starting_position, 193, -300, -121 \Rx:=-14.2, \Ry:=10.2, \Rz:=0), v200, z200, Tooldata_7;
MoveJ RelTool (starting_position, 195, -300, -122 \Rx:=-14.5, \Ry:=10.8, \Rz:=0), v200, z200, Tooldata_7;
MoveJ RelTool (starting_position, 197, -300, -123 \Rx:=-14.8, \Ry:=11.1, \Rz:=0), v200, z200, Tooldata_7;
MoveJ RelTool (starting_position, 199, -300, -125 \Rx:=-15.1, \Ry:=11.4, \Rz:=0), v200, z200, Tooldata_7;
MoveJ RelTool (starting_position, 201, -300, -126 \Rx:=-15.3, \Ry:=11.7, \Rz:=0), v200, z200, Tooldata_7;
MoveJ RelTool (starting_position, 203, -300, -128 \Rx:=-15.5, \Ry:=12, \Rz:=0), v200, z200, Tooldata_7;
MoveJ RelTool (starting_position, 205, -300, -129 \Rx:=-15.7, \Ry:=12.3, \Rz:=0), v200, z200, Tooldata_7;
MoveJ RelTool (starting_position, 206, -300, -131 \Rx:=-15.7, \Ry:=12.6, \Rz:=0), v200, z200, Tooldata_7;
MoveJ RelTool (starting_position, 208, -300, -133 \Rx:=-15.8, \Ry:=12.9, \Rz:=0), v200, z200, Tooldata_7;
MoveJ RelTool (starting_position, 209, -300, -134 \Rx:=-15.9, \Ry:=13.2, \Rz:=0), v200, z200, Tooldata_7;
MoveJ RelTool (starting_position, 209, -300, -136 \Rx:=-15.9, \Ry:=13.2, \Rz:=0), v200, z200, Tooldata_7;
MoveJ RelTool (starting_position, 210, -300, -138 \Rx:=-15.9, \Ry:=13.2, \Rz:=0), v200, z200, Tooldata_7;
MoveJ RelTool (starting_position, 210, -300, -140 \Rx:=-15.9, \Ry:=13.2, \Rz:=0), v200, z200, Tooldata_7;
MoveJ RelTool (starting_position, 210, -300, -142 \Rx:=-15.8, \Ry:=13.2, \Rz:=0), v200, z200, Tooldata_7;
MoveJ RelTool (starting_position, 210, -300, -144 \Rx:=-15.8, \Ry:=13.2, \Rz:=0), v200, z200, Tooldata_7;
MoveJ RelTool (starting_position, 209, -300, -146 \Rx:=-15.7, \Ry:=13.2, \Rz:=0), v200, z200, Tooldata_7;
MoveJ RelTool (starting_position, 208, -300, -148 \Rx:=-15.6, \Ry:=12.9, \Rz:=0), v200, z200, Tooldata_7;
MoveJ RelTool (starting_position, 207, -300, -151 \Rx:=-15.5, \Ry:=12.9, \Rz:=0), v200, z200, Tooldata_7;
MoveJ RelTool (starting_position, 206, -300, -153 \Rx:=-15.4, \Ry:=12.6, \Rz:=0), v200, z200, Tooldata_7;
MoveJ RelTool (starting_position, 204, -300, -155 \Rx:=-15.2, \Ry:=12.3, \Rz:=0), v200, z200, Tooldata_7;
MoveJ RelTool (starting_position, 202, -300, -158 \Rx:=-15.1, \Ry:=12, \Rz:=0), v200, z200, Tooldata_7;
MoveJ RelTool (starting_position, 200, -300, -160 \Rx:=-15, \Ry:=11.7, \Rz:=0), v200, z200, Tooldata_7;
MoveJ RelTool (starting_position, 197, -300, -162 \Rx:=-14.9, \Ry:=11.1, \Rz:=0), v200, z200, Tooldata_7;
MoveJ RelTool (starting_position, 194, -300, -165 \Rx:=-14.8, \Ry:=10.5, \Rz:=0), v200, z200, Tooldata_7;
MoveJ RelTool (starting_position, 191, -300, -167 \Rx:=-14.6, \Ry:=9.9, \Rz:=0), v200, z200, Tooldata_7;
MoveJ RelTool (starting_position, 188, -300, -169 \Rx:=-14.5, \Ry:=9.3, \Rz:=0), v200, z200, Tooldata_7;
MoveJ RelTool (starting_position, 184, -300, -171 \Rx:=-14.4, \Ry:=8.7, \Rz:=0), v200, z200, Tooldata_7;
MoveJ RelTool (starting_position, 180, -300, -173 \Rx:=-14.3, \Ry:=8.1, \Rz:=0), v200, z200, Tooldata_7;
MoveJ RelTool (starting_position, 177, -300, -175 \Rx:=-14.2, \Ry:=7.5, \Rz:=0), v200, z200, Tooldata_7;
MoveJ RelTool (starting_position, 173, -300, -176 \Rx:=-14.1, \Ry:=6.9, \Rz:=0), v200, z200, Tooldata_7;
MoveJ RelTool (starting_position, 169, -300, -178 \Rx:=-14, \Ry:=6, \Rz:=0), v200, z200, Tooldata_7;
MoveJ RelTool (starting_position, 165, -300, -179 \Rx:=-14, \Ry:=5.4, \Rz:=0), v200, z200, Tooldata_7;
MoveJ RelTool (starting_position, 160, -300, -180 \Rx:=-13.9, \Ry:=4.5, \Rz:=0), v200, z200, Tooldata_7;
MoveJ RelTool (starting_position, 156, -300, -181 \Rx:=-13.8, \Ry:=3.9, \Rz:=0), v200, z200, Tooldata_7;
MoveJ RelTool (starting_position, 151, -300, -181 \Rx:=-13.7, \Ry:=3, \Rz:=0), v200, z200, Tooldata_7;
MoveJ RelTool (starting_position, 147, -300, -182 \Rx:=-13.7, \Ry:=2.1, \Rz:=0), v200, z200, Tooldata_7;
MoveJ RelTool (starting_position, 143, -300, -182 \Rx:=-13.7, \Ry:=1.5, \Rz:=0), v200, z200, Tooldata_7;
MoveJ RelTool (starting_position, 139, -300, -182 \Rx:=-13.7, \Ry:=0.9, \Rz:=0), v200, z200, Tooldata_7;
MoveJ RelTool (starting_position, 135, -300, -182 \Rx:=-13.6, \Ry:=0.3, \Rz:=0), v200, z200, Tooldata_7;
MoveJ RelTool (starting_position, 131, -300, -181 \Rx:=-13.6, \Ry:=-0.6, \Rz:=0), v200, z200, Tooldata_7;
MoveJ RelTool (starting_position, 127, -300, -181 \Rx:=-13.6, \Ry:=-1.2, \Rz:=0), v200, z200, Tooldata_7;
MoveJ RelTool (starting_position, 124, -300, -180 \Rx:=-13.6, \Ry:=-1.8, \Rz:=0), v200, z200, Tooldata_7;
MoveJ RelTool (starting_position, 120, -300, -180 \Rx:=-13.6, \Ry:=-2.4, \Rz:=0), v200, z200, Tooldata_7;
MoveJ RelTool (starting_position, 117, -300, -179 \Rx:=-13.6, \Ry:=-3, \Rz:=0), v200, z200, Tooldata_7;
MoveJ RelTool (starting_position, 114, -300, -178 \Rx:=-13.6, \Ry:=-3.6, \Rz:=0), v200, z200, Tooldata_7;
MoveJ RelTool (starting_position, 111, -300, -178 \Rx:=-13.6, \Ry:=-3.9, \Rz:=0), v200, z200, Tooldata_7;
MoveJ RelTool (starting_position, 109, -300, -177 \Rx:=-13.6, \Ry:=-4.5, \Rz:=0), v200, z200, Tooldata_7;
MoveJ RelTool (starting_position, 107, -300, -176 \Rx:=-13.6, \Ry:=-4.8, \Rz:=0), v200, z200, Tooldata_7;
MoveJ RelTool (starting_position, 105, -300, -175 \Rx:=-13.5, \Ry:=-5.1, \Rz:=0), v200, z200, Tooldata_7;
MoveJ RelTool (starting_position, 103, -300, -174 \Rx:=-13.5, \Ry:=-5.4, \Rz:=0), v200, z200, Tooldata_7;
MoveJ RelTool (starting_position, 101, -300, -173 \Rx:=-13.4, \Ry:=-5.7, \Rz:=0), v200, z200, Tooldata_7;
MoveJ RelTool (starting_position, 100, -300, -172 \Rx:=-13.2, \Ry:=-6, \Rz:=0), v200, z200, Tooldata_7;
MoveJ RelTool (starting_position, 99, -300, -171 \Rx:=-13, \Ry:=-6, \Rz:=0), v200, z200, Tooldata_7;
MoveJ RelTool (starting_position, 97, -300, -170 \Rx:=-12.8, \Ry:=-6.3, \Rz:=0), v200, z200, Tooldata_7;
MoveJ RelTool (starting_position, 96, -300, -169 \Rx:=-12.5, \Ry:=-6.6, \Rz:=0), v200, z200, Tooldata_7;
MoveJ RelTool (starting_position, 96, -300, -168 \Rx:=-12.2, \Ry:=-6.6, \Rz:=0), v200, z200, Tooldata_7;
MoveJ RelTool (starting_position, 95, -300, -168 \Rx:=-11.9, \Ry:=-6.9, \Rz:=0), v200, z200, Tooldata_7;
MoveJ RelTool (starting_position, 94, -300, -167 \Rx:=-11.5, \Ry:=-6.9, \Rz:=0), v200, z200, Tooldata_7;
MoveJ RelTool (starting_position, 94, -300, -166 \Rx:=-11, \Ry:=-6.9, \Rz:=0), v200, z200, Tooldata_7;
MoveJ RelTool (starting_position, 94, -300, -165 \Rx:=-10.5, \Ry:=-6.9, \Rz:=0), v200, z200, Tooldata_7;
MoveJ RelTool (starting_position, 94, -300, -165 \Rx:=-9.9, \Ry:=-6.9, \Rz:=0), v200, z200, Tooldata_7;
MoveJ RelTool (starting_position, 93, -300, -164 \Rx:=-9.4, \Ry:=-6.9, \Rz:=0), v200, z200, Tooldata_7;
MoveJ RelTool (starting_position, 93, -300, -163 \Rx:=-8.8, \Ry:=-7.2, \Rz:=0), v200, z200, Tooldata_7;
MoveJ RelTool (starting_position, 92, -300, -163 \Rx:=-8.2, \Ry:=-7.2, \Rz:=0), v200, z200, Tooldata_7;
MoveJ RelTool (starting_position, 92, -300, -162 \Rx:=-7.6, \Ry:=-7.2, \Rz:=0), v200, z200, Tooldata_7;
MoveJ RelTool (starting_position, 92, -300, -161 \Rx:=-7, \Ry:=-7.2, \Rz:=0), v200, z200, Tooldata_7;
MoveJ RelTool (starting_position, 92, -300, -161 \Rx:=-6.4, \Ry:=-7.5, \Rz:=0), v200, z200, Tooldata_7;
MoveJ RelTool (starting_position, 92, -300, -160 \Rx:=-5.9, \Ry:=-7.5, \Rz:=0), v200, z200, Tooldata_7;
MoveJ RelTool (starting_position, 92, -300, -160 \Rx:=-5.3, \Ry:=-7.2, \Rz:=0), v200, z200, Tooldata_7;
MoveJ RelTool (starting_position, 92, -300, -159 \Rx:=-4.8, \Ry:=-7.2, \Rz:=0), v200, z200, Tooldata_7;
MoveJ RelTool (starting_position, 92, -300, -158 \Rx:=-4.2, \Ry:=-7.2, \Rz:=0), v200, z200, Tooldata_7;
MoveJ RelTool (starting_position, 92, -300, -158 \Rx:=-3.7, \Ry:=-7.2, \Rz:=0), v200, z200, Tooldata_7;
MoveJ RelTool (starting_position, 92, -300, -157 \Rx:=-3.2, \Ry:=-7.2, \Rz:=0), v200, z200, Tooldata_7;
MoveJ RelTool (starting_position, 92, -300, -156 \Rx:=-2.7, \Ry:=-7.2, \Rz:=0), v200, z200, Tooldata_7;
MoveJ RelTool (starting_position, 92, -300, -156 \Rx:=-2.4, \Ry:=-7.2, \Rz:=0), v200, z200, Tooldata_7;
MoveJ RelTool (starting_position, 92, -300, -155 \Rx:=-1.9, \Ry:=-7.2, \Rz:=0), v200, z200, Tooldata_7;
MoveJ RelTool (starting_position, 92, -300, -154 \Rx:=-1.5, \Ry:=-7.2, \Rz:=0), v200, z200, Tooldata_7;
MoveJ RelTool (starting_position, 92, -300, -154 \Rx:=-1.1, \Ry:=-7.2, \Rz:=0), v200, z200, Tooldata_7;
MoveJ RelTool (starting_position, 92, -300, -153 \Rx:=-0.7, \Ry:=-7.2, \Rz:=0), v200, z200, Tooldata_7;
MoveJ RelTool (starting_position, 92, -300, -152 \Rx:=-0.3, \Ry:=-7.2, \Rz:=0), v200, z200, Tooldata_7;
MoveJ RelTool (starting_position, 92, -300, -152 \Rx:=0, \Ry:=-7.2, \Rz:=0), v200, z200, Tooldata_7;
MoveJ RelTool (starting_position, 92, -300, -151 \Rx:=0.4, \Ry:=-7.2, \Rz:=0), v200, z200, Tooldata_7;
MoveJ RelTool (starting_position, 92, -300, -150 \Rx:=0.7, \Ry:=-7.2, \Rz:=0), v200, z200, Tooldata_7;
MoveJ RelTool (starting_position, 92, -300, -149 \Rx:=1, \Ry:=-7.2, \Rz:=0), v200, z200, Tooldata_7;
MoveJ RelTool (starting_position, 92, -300, -149 \Rx:=1.3, \Ry:=-7.2, \Rz:=0), v200, z200, Tooldata_7;
MoveJ RelTool (starting_position, 92, -300, -148 \Rx:=1.6, \Ry:=-7.2, \Rz:=0), v200, z200, Tooldata_7;
MoveJ RelTool (starting_position, 92, -300, -147 \Rx:=1.8, \Ry:=-7.2, \Rz:=0), v200, z200, Tooldata_7;
MoveJ RelTool (starting_position, 92, -300, -146 \Rx:=2.1, \Ry:=-7.2, \Rz:=0), v200, z200, Tooldata_7;
MoveJ RelTool (starting_position, 92, -300, -145 \Rx:=2.2, \Ry:=-7.2, \Rz:=0), v200, z200, Tooldata_7;
MoveJ RelTool (starting_position, 92, -300, -145 \Rx:=2.4, \Ry:=-7.2, \Rz:=0), v200, z200, Tooldata_7;
MoveJ RelTool (starting_position, 93, -300, -144 \Rx:=2.5, \Ry:=-7.2, \Rz:=0), v200, z200, Tooldata_7;
MoveJ RelTool (starting_position, 93, -300, -143 \Rx:=2.6, \Ry:=-7.2, \Rz:=0), v200, z200, Tooldata_7;
MoveJ RelTool (starting_position, 93, -300, -142 \Rx:=2.6, \Ry:=-6.9, \Rz:=0), v200, z200, Tooldata_7;
MoveJ RelTool (starting_position, 94, -300, -141 \Rx:=2.7, \Ry:=-6.9, \Rz:=0), v200, z200, Tooldata_7;
MoveJ RelTool (starting_position, 94, -300, -141 \Rx:=2.7, \Ry:=-6.9, \Rz:=0), v200, z200, Tooldata_7;
MoveJ RelTool (starting_position, 95, -300, -140 \Rx:=2.7, \Ry:=-6.9, \Rz:=0), v200, z200, Tooldata_7;
MoveJ RelTool (starting_position, 95, -300, -139 \Rx:=2.7, \Ry:=-6.6, \Rz:=0), v200, z200, Tooldata_7;
MoveJ RelTool (starting_position, 95, -300, -138 \Rx:=2.7, \Ry:=-6.6, \Rz:=0), v200, z200, Tooldata_7;
MoveJ RelTool (starting_position, 96, -300, -137 \Rx:=2.7, \Ry:=-6.6, \Rz:=0), v200, z200, Tooldata_7;
MoveJ RelTool (starting_position, 96, -300, -137 \Rx:=2.7, \Ry:=-6.6, \Rz:=0), v200, z200, Tooldata_7;
MoveJ RelTool (starting_position, 96, -300, -136 \Rx:=2.7, \Ry:=-6.6, \Rz:=0), v200, z200, Tooldata_7;
MoveJ RelTool (starting_position, 97, -300, -135 \Rx:=2.7, \Ry:=-6.3, \Rz:=0), v200, z200, Tooldata_7;
MoveJ RelTool (starting_position, 98, -300, -134 \Rx:=2.8, \Ry:=-6.3, \Rz:=0), v200, z200, Tooldata_7;
MoveJ RelTool (starting_position, 99, -300, -134 \Rx:=2.8, \Ry:=-6, \Rz:=0), v200, z200, Tooldata_7;
MoveJ RelTool (starting_position, 100, -300, -133 \Rx:=3, \Ry:=-6, \Rz:=0), v200, z200, Tooldata_7;
MoveJ RelTool (starting_position, 100, -300, -132 \Rx:=3.1, \Ry:=-5.7, \Rz:=0), v200, z200, Tooldata_7;
MoveJ RelTool (starting_position, 101, -300, -132 \Rx:=3.3, \Ry:=-5.7, \Rz:=0), v200, z200, Tooldata_7;
MoveJ RelTool (starting_position, 102, -300, -131 \Rx:=3.4, \Ry:=-5.4, \Rz:=0), v200, z200, Tooldata_7;
MoveJ RelTool (starting_position, 103, -300, -130 \Rx:=3.6, \Ry:=-5.4, \Rz:=0), v200, z200, Tooldata_7;
MoveJ RelTool (starting_position, 103, -300, -130 \Rx:=3.8, \Ry:=-5.4, \Rz:=0), v200, z200, Tooldata_7;
MoveJ RelTool (starting_position, 104, -300, -129 \Rx:=4, \Ry:=-5.1, \Rz:=0), v200, z200, Tooldata_7;
MoveJ RelTool (starting_position, 105, -300, -129 \Rx:=4.2, \Ry:=-4.8, \Rz:=0), v200, z200, Tooldata_7;
MoveJ RelTool (starting_position, 106, -300, -128 \Rx:=4.5, \Ry:=-4.8, \Rz:=0), v200, z200, Tooldata_7;
MoveJ RelTool (starting_position, 107, -300, -128 \Rx:=4.9, \Ry:=-4.5, \Rz:=0), v200, z200, Tooldata_7;
MoveJ RelTool (starting_position, 108, -300, -128 \Rx:=5.2, \Ry:=-4.5, \Rz:=0), v200, z200, Tooldata_7;
MoveJ RelTool (starting_position, 108, -300, -127 \Rx:=5.6, \Ry:=-4.5, \Rz:=0), v200, z200, Tooldata_7;
MoveJ RelTool (starting_position, 109, -300, -127 \Rx:=6, \Ry:=-4.2, \Rz:=0), v200, z200, Tooldata_7;
MoveJ RelTool (starting_position, 110, -300, -127 \Rx:=6.3, \Ry:=-4.2, \Rz:=0), v200, z200, Tooldata_7;
MoveJ RelTool (starting_position, 111, -300, -126 \Rx:=6.6, \Ry:=-3.9, \Rz:=0), v200, z200, Tooldata_7;
MoveJ RelTool (starting_position, 111, -300, -126 \Rx:=6.9, \Ry:=-3.9, \Rz:=0), v200, z200, Tooldata_7;
MoveJ RelTool (starting_position, 112, -300, -126 \Rx:=7.2, \Ry:=-3.9, \Rz:=0), v200, z200, Tooldata_7;
MoveJ RelTool (starting_position, 113, -300, -126 \Rx:=7.4, \Ry:=-3.6, \Rz:=0), v200, z200, Tooldata_7;
MoveJ RelTool (starting_position, 113, -300, -125 \Rx:=7.6, \Ry:=-3.6, \Rz:=0), v200, z200, Tooldata_7;
MoveJ RelTool (starting_position, 114, -300, -125 \Rx:=7.8, \Ry:=-3.3, \Rz:=0), v200, z200, Tooldata_7;
MoveJ RelTool (starting_position, 115, -300, -125 \Rx:=7.9, \Ry:=-3.3, \Rz:=0), v200, z200, Tooldata_7;
MoveJ RelTool (starting_position, 116, -300, -125 \Rx:=7.9, \Ry:=-3, \Rz:=0), v200, z200, Tooldata_7;
MoveJ RelTool (starting_position, 116, -300, -124 \Rx:=7.9, \Ry:=-3, \Rz:=0), v200, z200, Tooldata_7;
